(* CoDeSys 2.3 project: DPC_TM10.pro *)
(* Libraries: BODAS-design_Library_V20.lib 15.2.18 10:15:14, BODAS_RC28-14_30_Family_V01_03.lib 7.6.18 09:26:32, CIA405_Library_V02_01.lib 15.2.18 10:15:14, INEXT_Library_V01_06.lib 15.2.18 10:15:14, lib_mat.lib 15.2.18 10:15:14, RCE_InitParameter_V01_03.lib 15.2.18 10:15:14, RCE_Library_V01_03.lib 15.2.18 10:15:14, SAFOUT_Library_V02_04.lib 15.2.18 10:15:14, STANDARD_V02_00.lib 15.2.18 10:15:14, Util.lib 13.6.14 15:20:40 *)

(* Global variable list: Global_CONST *)
VAR_GLOBAL CONSTANT
	LID_DefaultSession_DU8       : USINT      := 16#7F;
	LID_DemoSession_DU8         : USINT      := 16#80;
	LID_ServiceSession_DU8      : USINT      := 16#91;
    LID_AdjustmentSession_DU8    : USINT     := 16#B3;
    LID_Adjustment1Session_DU8   : USINT     := 16#C1;
    LID_Adjustment2Session_DU8    : USINT     := 16#C2;
    LID_Adjustment3Session_DU8    : USINT    := 16#C3;
    LID_Adjustment4Session_DU8    : USINT     := 16#C4;
    LID_DevelopmentSession_DU8   : USINT     := 16#F7;


	CYCLE							: USINT	:= 10;		(* cycle time of the main task *)
	MAIN_TASK_PRIO				: BYTE	:= 100;		(*priority of the main task*)
	SIMU_motSpeed_b8			: BOOL	:= FALSE;

	DST_JOY						: INT		:= 1;			(* Type of the Drive joystick *)
	GESSMAN						: INT 	:= 0;			(* Type of the Drive joystick *)

	ST_RANGE						: INT		:= 1000;
	PAGE1_OFFSET				: INT 	:= 256;
	PAGE2_OFFSET				: INT 	:= 512;

	DELAY_STANDARD				: UINT	:= 600; 		(* increased for Fair !!! *)
	DEBOUNCE_FOR_SAVOUT		: UINT	:= 200;
	MAX_LIMIT_SPEED_MUL1000	: INT		:= 1800;
	(*LIMIT_SPEED_1_MUL1000	: INT 	:=	400;*)

	POTI_CURRENT_ERR_MIN		: INT		:= 700;		(* Unit = uA *)
	POTI_CURRENT_ERR_MAX		: INT		:= 1200;		(* Unit = uA *)

	KPDv							: REAL	:= 0.95; 	(* Volumetric efficiency *)
	(*iReductor_1					: REAL	:= 0.792;	(* передачное число редуктора МП19-4240010 *)*)

	V_TRANSM_BORDER			: INT		:= 500;		(* Граница, после которой включаются в работу моторы *)
	(*CAN1_MESSAGE_FREQ			: UINT	:= 100;		(* Промежуток между отправками посылок в шину, ms *)*)
	CYCLES_FOR_CAN_SEND		: INT		:= 10;

	Pi								: REAL	:= 3.14;		(* Число Пи *)
(******************** Definition:   PWM output - High side  *******************)
(******************************************************************************)
	POH_CL_DEBOUNCE			: UINT	:= 100;				(* debounce time [ms] for error detection *)
	POH_CL_DITHER_FREQUENCY	: UINT	:= f_100Hz_DU16;	(* dither frequency [Hz]*)
	POH_CL_RESISTANCE_MIN	: UDINT	:= 2000; 			(* min resistance of solenoid for error detection [mOhm]*)
	POH_CL_RESISTANCE_MAX	: UDINT	:= 52000;			(* max resistance of solenoid for error detection[mOhm] *)
	POH_CL_KP					: UINT	:= 250;				(*Kp factor*)
	POH_CL_KI					: UINT 	:= 250;				(*Ki factor*)
(******************** Definition:   PWM output - Low side - FAN_Drive *********)
(******************************************************************************)
	POL_CL_DEBOUNCE			: UINT	:= 100;				(* debounce time [ms] for error detection *)
	POL_CL_DITHER_FREQUENCY	: UINT	:= f_100Hz_DU16;	(* dither frequency [Hz]*)
	POL_CL_RESISTANCE_MIN	: UDINT	:= 2000; 			(* min resistance of solenoid for error detection [mOhm]*)
	POL_CL_RESISTANCE_MAX	: UDINT	:= 52000;			(* max resistance of solenoid for error detection[mOhm] *)
	POL_CL_KP					: UINT 	:= 250;				(*Kp factor*)
	POL_CL_KI					: UINT 	:= 250;				(*Ki factor*)
(******************************************************************************)
(******************** Definition:   Digital output - High side  ***************)
(******************************************************************************)
	DOH_DEBOUNCE				: UINT	:= 200;				(* debounce time [ms] for error detection *)
	DOH_DITHER_FREQUENCY		: UINT	:= f_100Hz_DU16;	(* dither frequency [Hz]*)
	DOH_RESISTANCE_MIN		: UDINT	:= 6000;				(* min resistance of solenoid for error detection [mOhm]*)
	DOH_RESISTANCE_MAX		: UDINT	:= 44000;			(* max resistance of solenoid for error detection[mOhm] *)
	DOH_WORKING_ARM_MAX		: UDINT	:= 60000;			(* Для плеч гидрораспределителя *)
	MS_IN_MINUTE				: DINT	:= 60000;

	AOV_DITHER_FREQUENCY		: UINT	:= f_100Hz_DU16;	(* dither frequency [Hz]*)

	MAX_VOLTAGE_FOR_JOY		: INT := 5000; (* Максимальное напряжение для джойстиков, мВ *)

	PWM_MODE						: INT		:= 0;					(* Режим ШИМ-выхода без поддержания тока *)
	PWM_CURRENT_MODE			: INT		:= 1;					(* Режим ШИМ-выхода с обратной связью по току *)

	AOC_MODE						: INT		:= 0;					(* Analog Output Current *)
	AOV_MODE						: INT		:= 1;					(* Analog Output Voltage *)

END_VAR

(* Global variable list: Globale_Variablen *)
VAR_GLOBAL
	para_s	: para_ts;				(* structure for the storage of the parameter *)
	err		: applError_ts;		(* structure for the error management *)
	CAN_s		: struc_Can;			(* structure for the CAN bus management *)
	J1939_s	: struc_J1939;
	IO_Chnl	: struc_IO_Chnl;		(* structure for the channels of the inputs and the outputs *)
	output	: struc_outputs;
	input		: struc_inputs;
	Uds_s    : struc_Uds;


(***********************************************************************************)
	j1939_DIESEL_DM1_s 	: j1939_dtcList_ts;
	j1939_DIESEL_DM2_s 	: j1939_dtcList_ts;
(***********************************************************************************)
	hydroDist_debounce			: UINT;				(* debounce time [ms] for error detection *)
	hydroDist_frequency			: UINT;				(* dither frequency [Hz]*)
	hydroDist_resistance_min	: UDINT; 			(* min resistance of solenoid for error detection [mOhm]*)
	hydroDist_resistance_max	: UDINT;				(* max resistance of solenoid for error detection[mOhm] *)
	hydroDist_kp_1					: UINT;				(*Kp factor*)
	hydroDist_kp_2					: UINT;				(*Kp factor*)
	hydroDist_ki_1					: UINT;				(*Ki factor*)
	hydroDist_ki_2					: UINT;				(*Ki factor*)

END_VAR

(* Global variable list: State_Machines *)
VAR_GLOBAL
	stMachine_s16				: INT		:= 0;		(*	machine state 	*)
	stStartlock_b8				: BOOL; 				(* No HW problems detected at start, if TRUE *)
	stStartAppl_b8				: BOOL;				(* Application Start condition OK, if TRUE *)
END_VAR

VAR_GLOBAL CONSTANT

(*************************************************************************************************)
	DEACTIVATED				:	INT	:=	0;
	ACTIVATED				:	INT	:=	1;

END_VAR

(* Data type in Enums *)
TYPE applError_e:
(*********************************************)
(*  DON'T MAKE ANY CHANGES TO THIS ENUMS!!   *)
(*     FILE WAS AUTOMATICALLY GENERATED!!    *)
(*********************************************)
(

   ERR_FIRST_CODE                       := 16#8000,
   ERR_CAN_DIAG                         := 16#8001,
   ERR_PWRON_SUPPLY_VB_LOW              := 16#8036,
   ERR_PWRON_SUPPLY_VSS                 := 16#8037,
   ERR_PWRON_HWMONITOR_1                := 16#8038,
   ERR_PWRON_STARTCONDITION_1           := 16#8039,
   ERR_PWRON_ENGINE_SPEED               := 16#8040,
   ERR_PWRON_HWMONITOR_2                := 16#8041,
   ERR_PWRON_STARTCONDITION_2           := 16#8042,
   ERR_PWRON_SAFOUT_CABLE_BRAKE         := 16#8043,
   ERR_PWRON_SAFOUT_SHORT_CIRCUIT       := 16#8044,
   ERR_PWRON_POWERSWITCH_1              := 16#8045,
   ERR_PWRON_POWERSUPPLY                := 16#8046,
   ERR_PWRON_POWERSWITCH_2              := 16#8047,
   ERR_PWRON_REVERSE_POWER              := 16#8048,
   ERR_PWRON_EMERGENCY_STOP             := 16#8049,
   ERR_SUPPLY_VB_HIGH                   := 16#8031,
   ERR_SUPPLY_VB_LOW                    := 16#8032,
   ERR_SUPPLY_VSS1                      := 16#8033,
   ERR_SUPPLY_VSS2                      := 16#8034,
   ERR_LAST_CODE                        := 16#8099

);
END_TYPE

(* Data type in Structures *)
TYPE applError_ts:
(***********************************************)
(*  DON'T MAKE ANY CHANGES TO THIS STRUCTURE!! *)
(*      FILE WAS AUTOMATICALLY GENERATED!!     *)
(***********************************************)
STRUCT

   First_code_b8                    : BOOL;
   Can_diag_b8                      : BOOL;
   Pwron_supply_vb_low_b8           : BOOL;
   Pwron_supply_vss_b8              : BOOL;
   Pwron_hwmonitor_1_b8             : BOOL;
   Pwron_startcondition_1_b8        : BOOL;
   Pwron_engine_speed_b8            : BOOL;
   Pwron_hwmonitor_2_b8             : BOOL;
   Pwron_startcondition_2_b8        : BOOL;
   Pwron_safout_cable_brake_b8      : BOOL;
   Pwron_safout_short_circuit_b8    : BOOL;
   Pwron_powerswitch_1_b8           : BOOL;
   Pwron_powersupply_b8             : BOOL;
   Pwron_powerswitch_2_b8           : BOOL;
   Pwron_reverse_power_b8           : BOOL;
   Pwron_emergency_stop_b8          : BOOL;
   Supply_vb_high_b8                : BOOL;
   Supply_vb_low_b8                 : BOOL;
   Supply_vss1_b8                   : BOOL;
   Supply_vss2_b8                   : BOOL;
   Last_code_b8                     : BOOL;

END_STRUCT
END_TYPE

(* Data type in Diag/Error *)
TYPE ApplErrorNew_ts :
(* ApplError_ts *)
STRUCT
	Code_u16					: UINT;
	Description_as8		: STRING(32);
(*	Description_as8		: ARRAY [1..4] OF STRING(32);*)
END_STRUCT
END_TYPE

(* Data type in Diag/Parameter *)
TYPE attr1_tu :
STRUCT
	MinValue_s16		: INT;
(*
	InputChannel_u16	: UINT;
	ListNumber_u16		: UINT;
	data_au8 			: ARRAY [1..2] OF USINT;
*)
END_STRUCT
END_TYPE

(* Data type in Diag/Parameter *)
TYPE attr2_tu :
STRUCT
	MaxValue_s16		: INT;
(*
	InputChannel_u16	: UINT;
	ListEntries_u16	: UINT;
	data_au8 			: ARRAY [1..2] OF USINT;
*)
END_STRUCT
END_TYPE

(* Data type in Diag/Parameter *)
TYPE attr3_tu :
STRUCT
	StepWidth_u16			: UINT;
(*
	FunctionNumber_u16	: UINT;
	FrequencyRange_u16	: UINT;
	data_au8 				: ARRAY [1..2] OF USINT;
*)
END_STRUCT
END_TYPE

(* Data type in Diag/Parameter *)
TYPE attr4_tu :
STRUCT
	DefaultValue_as16		: INT;
(*
	DefaultValue_as16		: ARRAY [1..16] OF INT;
	AnalogChannel_as16	: ARRAY [1..16] OF INT;
	Frequency_as16			: ARRAY [1..16] OF INT;
	data_au8 				: ARRAY [1..2] OF USINT;
*)
END_STRUCT
END_TYPE

(* Data type in Diag/Parameter *)
TYPE attr_tu :
STRUCT
	NumberOfDigits_u16	: UINT;
	BargraphMaximum_u16	: UINT;
	PostCommaDigits_u16	: UINT;
	data_au8 				: ARRAY [1..2] OF USINT;
END_STRUCT
END_TYPE

(* Data type in Diag/Parameter *)
TYPE EEPROMAdrress_ts :
STRUCT
	Page_u8		: USINT;
	IntIndex_u8	: USINT;
END_STRUCT
END_TYPE

(* Data type in 20_CAN *)
TYPE enum_Can :
	(
		CAN_RESET_STOP		:= 0,
		CAN_RESET_START	:= 1,
		CAN_RESET_WAIT		:= 2
	);
END_TYPE

(* Data type in 40_Other *)
TYPE enum_Startlock_Test :
(
	(* startlock tests *)
	TEST_SUPPLY	:= 1,
	TEST_VSS1,
	TEST_VSS2,
	TEST_VSS3,
	TEST_HWMONITOR_1,
	TEST_CONDITION_1,
	TEST_SWITCH1,
	TEST_SWITCH2,
	TEST_SAFOUT,
	TEST_DIESEL,
	TEST_HWMONITOR_2,
	TEST_CONDITION_2,
	TEST_MAX
);
END_TYPE

(* Data type in Diag/Error *)
TYPE ErrorEntry_ts :
STRUCT
	Code_u16					: UINT;
	Param_u8					: USINT;
	Frequency_u8			: USINT;
	TimeStamp_u32			: UDINT;
END_STRUCT
END_TYPE

(* Data type in Diag/Other *)
TYPE FuncParams_ts :
STRUCT
	Description_as8		: STRING(32);
(*	Description_as8		: ARRAY [1..4] OF STRING(32);*)
END_STRUCT
END_TYPE

(* Data type in Enums *)
TYPE para_e:
(*********************************************)
(*  DON'T MAKE ANY CHANGES TO THIS ENUMS!!   *)
(*    FILE WAS AUTOMATICALLY GENERATED!!     *)
(*********************************************)
(

(* Menu 1 *)

(* Basic *)
   EEP_number_1_1_1_e:= 790,      (* 0  (0 - 2) *)
   EEP_Input_to_Output_Mode_e:= 770,(* Not Active  (0 - 2) *)
   EEP_test_par_new_e:= 773,      (* Not Active  (0 - 2) *)
   EEP_test_params_e:= 771,       (* Not Active  (0 - 2) *)
   EEP_test_par2_e:= 772,         (* Not Active  (0 - 2) *)

(* Test Type *)
   EEP_Trimming_type_e:= 818,     (* 53  (0 - 511) *)
   EEP_Analog_type_e:= 819,       (* 245  (53 - ) *)
   EEP_Curve_Type_e:= 820,        (* 245  (66 - 67) *)
   EEP_Function_Type_e:= 821,     (* 248  (248 - 254) *)
   EEP_Percent_Type_e:= 822,      (* 0 % (0 - 1000) *)
   EEP_Ramp_Type_e:= 823,         (* 0 % (0 - 100) *)
   EEP_Switch_Type_e:= 824,       (* 1  ( - ) *)
   EEP_List_Type_e:= 825,         (* AOC  (3 - 2) *)

(* Test Number *)
   EEP_number_1_3_1_e:= 782,      (* 0 ms (0 - 30000) *)
   EEP_number_1_3_2_e:= 783,      (* 0 ms (0 - 30000) *)
   EEP_number_1_3_3_e:= 784,      (* 0 ms (0 - 30000) *)
   EEP_number_1_3_4_e:= 785,      (* 0 ms (0 - 30000) *)
   EEP_number_1_3_5_e:= 786,      (* 0 ms (0 - 30000) *)
   EEP_number_1_3_6_e:= 787,      (* 0 ms (0 - 30000) *)
   EEP_number_1_3_7_e:= 788,      (* 0 ms (0 - 30000) *)
   EEP_number_1_3_8_e:= 789,      (* 0 ms (0 - 30000) *)


(* Menu 2 *)

(* Output Cfg 1-8 *)
   EEP_Out_Cfg_01_e:= 832,        (* PWM  (1 - 2) *)
   EEP_Out_Cfg_02_e:= 833,        (* PWM  (1 - 2) *)
   EEP_Out_Cfg_03_e:= 834,        (* PWM  (1 - 2) *)
   EEP_Out_Cfg_04_e:= 835,        (* PWM  (1 - 2) *)
   EEP_Out_Cfg_05_e:= 836,        (* PWM  (1 - 2) *)
   EEP_Out_Cfg_06_e:= 837,        (* PWM  (1 - 2) *)
   EEP_Out_Cfg_07_e:= 838,        (* PWM  (1 - 2) *)
   EEP_Out_Cfg_08_e:= 839,        (* PWM  (1 - 2) *)

(* Output Cfg 9-16 *)
   EEP_Out_Cfg_09_e:= 840,        (* PWM  (1 - 2) *)
   EEP_Out_Cfg_10_e:= 841,        (* PWM  (1 - 2) *)
   EEP_Out_Cfg_11_e:= 842,        (* PWM  (1 - 2) *)
   EEP_Out_Cfg_12_e:= 843,        (* PWM  (1 - 2) *)
   EEP_Out_Cfg_13_e:= 844,        (* PWM  (1 - 2) *)
   EEP_Out_Cfg_14_e:= 845,        (* PWM  (1 - 2) *)
   EEP_Out_Cfg_15_e:= 846,        (* PWM  (1 - 2) *)
   EEP_Out_Cfg_16_e:= 847,        (* PWM  (1 - 2) *)

(* Output Cfg 17-24 *)
   EEP_Out_Cfg_17_e:= 848,        (* PWM  (1 - 2) *)
   EEP_Out_Cfg_18_e:= 849,        (* PWM  (1 - 2) *)
   EEP_Out_Cfg_19_e:= 850,        (* Not Active  (0 - 2) *)
   EEP_Out_Cfg_20_e:= 851,        (* Not Active  (0 - 2) *)
   EEP_Out_Cfg_21_e:= 852,        (* Not Active  (0 - 2) *)
   EEP_Out_Cfg_22_e:= 853,        (* Not Active  (0 - 2) *)
   EEP_Out_Cfg_23_e:= 854,        (* Not Active  (0 - 2) *)
   EEP_Out_Cfg_24_e:= 855,        (* Not Active  (0 - 2) *)

(* Output Cfg 25-32 *)
   EEP_Out_Cfg_25_e:= 856,        (* Not Active  (0 - 2) *)
   EEP_Out_Cfg_26_e:= 857,        (* Not Active  (0 - 2) *)
   EEP_Out_Cfg_27_e:= 858,        (* Not Active  (0 - 2) *)
   EEP_Out_Cfg_28_e:= 859,        (* Not Active  (0 - 2) *)
   EEP_Out_Cfg_29_e:= 860,        (* Not Active  (0 - 2) *)
   EEP_Out_Cfg_30_e:= 861,        (* Not Active  (0 - 2) *)
   EEP_Out_Cfg_31_e:= 862,        (* Not Active  (0 - 2) *)
   EEP_Out_Cfg_32_e:= 863,        (* Not Active  (0 - 2) *)

(* Output Cfg 33-40 *)
   EEP_Out_Cfg_33_e:= 864,        (* PWM  (2 - 2) *)
   EEP_Out_Cfg_34_e:= 865,        (* PWM  (2 - 2) *)
   EEP_Out_Cfg_35_e:= 866,        (* PWM  (2 - 2) *)
   EEP_Out_Cfg_36_e:= 867,        (* PWM  (2 - 2) *)
   EEP_Out_Cfg_37_e:= 868,        (* PWM  (1 - 2) *)
   EEP_Out_Cfg_38_e:= 869,        (* PWM  (1 - 2) *)
   EEP_Out_Cfg_39_e:= 870,        (* PWM  (1 - 2) *)
   EEP_Out_Cfg_40_e:= 871,        (* PWM  (1 - 2) *)

(* Output Cfg 41-47 *)
   EEP_Out_Cfg_41_e:= 872,        (* PWM  (1 - 2) *)
   EEP_Out_Cfg_42_e:= 873,        (* PWM  (1 - 2) *)
   EEP_Out_Cfg_43_e:= 874,        (* PWM  (1 - 2) *)
   EEP_Out_Cfg_44_e:= 875,        (* PWM  (1 - 2) *)
   EEP_Out_Cfg_45_e:= 876,        (* PWM  (1 - 2) *)
   EEP_Out_Cfg_46_e:= 877,        (* PWM  (1 - 2) *)
   EEP_Out_Cfg_47_e:= 878,        (* AOV  (3 - 2) *)

(* AOV Configuration *)
   EEP_AOV_Debounce_e:= 880,      (* 200 ms (50 - 250) *)
   EEP_AOV_Freq_e:= 881,          (* 80  (0 - 5000) *)
   EEP_AOV_Res_Min_e:= 882,       (* 0 Ohm (0 - 3000) *)
   EEP_AOV_Res_Max_e:= 883,       (* 0 Ohm (0 - 3000) *)
   EEP_AOV_Kp_e:= 884,            (* 250  (0 - 2000) *)
   EEP_AOV_Ki_e:= 885,            (* 250  (0 - 500) *)

(* AOC Configuration *)
   EEP_AOC_Debounce_e:= 888,      (* 200 ms (50 - 250) *)
   EEP_AOC_Freq_e:= 889,          (* 5000  (0 - 5000) *)
   EEP_AOC_Res_Min_e:= 890,       (* 0 Ohm (0 - 3000) *)
   EEP_AOC_Res_Max_e:= 891,       (* 0 Ohm (0 - 3000) *)
   EEP_AOC_Kp_e:= 892,            (* 250  (0 - 2000) *)
   EEP_AOC_Ki_e:= 893,            (* 250  (0 - 500) *)


(* Menu 3 *)

(* Output Value 1-8 *)
   EEP_Out_Val_01_e:= 896,        (* 0 % / mA (0 - 10000) *)
   EEP_Out_Val_02_e:= 897,        (* 0 % / mA (0 - 10000) *)
   EEP_Out_Val_03_e:= 898,        (* 0 % / mA (0 - 10000) *)
   EEP_Out_Val_04_e:= 899,        (* 0 % / mA (0 - 10000) *)
   EEP_Out_Val_05_e:= 900,        (* 0 % / mA (0 - 10000) *)
   EEP_Out_Val_06_e:= 901,        (* 0 % / mA (0 - 10000) *)
   EEP_Out_Val_07_e:= 902,        (* 0 % / mA (0 - 10000) *)
   EEP_Out_Val_08_e:= 903,        (* 0 % / mA (0 - 10000) *)

(* Output Value 9-16 *)
   EEP_Out_Val_09_e:= 904,        (* 0 % / mA (0 - 10000) *)
   EEP_Out_Val_10_e:= 905,        (* 0 % / mA (0 - 10000) *)
   EEP_Out_Val_11_e:= 906,        (* 0 % / mA (0 - 10000) *)
   EEP_Out_Val_12_e:= 907,        (* 0 % / mA (0 - 10000) *)
   EEP_Out_Val_13_e:= 908,        (* 0 % / mA (0 - 10000) *)
   EEP_Out_Val_14_e:= 909,        (* 0 % / mA (0 - 10000) *)
   EEP_Out_Val_15_e:= 910,        (* 0 % / mA (0 - 10000) *)
   EEP_Out_Val_16_e:= 911,        (* 0 % / mA (0 - 10000) *)

(* Output Value 17-36 *)
   EEP_Out_Val_17_e:= 912,        (* 0 % / mA (0 - 10000) *)
   EEP_Out_Val_18_e:= 913,        (* 0 % / mA (0 - 10000) *)
   EEP_Out_Val_33_e:= 916,        (* 0 % / mA (0 - 10000) *)
   EEP_Out_Val_34_e:= 917,        (* 0 % / mA (0 - 10000) *)
   EEP_Out_Val_35_e:= 918,        (* 0 % / mA (0 - 10000) *)
   EEP_Out_Val_36_e:= 919,        (* 0 % / mA (0 - 10000) *)

(* Output Value 37-44 *)
   EEP_Out_Val_37_e:= 920,        (* 0 % / mA (0 - 10000) *)
   EEP_Out_Val_38_e:= 921,        (* 0 % / mA (0 - 10000) *)
   EEP_Out_Val_39_e:= 922,        (* 0 % / mA (0 - 10000) *)
   EEP_Out_Val_40_e:= 923,        (* 0 % / mA (0 - 10000) *)
   EEP_Out_Val_41_e:= 924,        (* 0 % / mA (0 - 10000) *)
   EEP_Out_Val_42_e:= 925,        (* 0 % / mA (0 - 10000) *)
   EEP_Out_Val_43_e:= 926,        (* 0 % / mA (0 - 10000) *)
   EEP_Out_Val_44_e:= 927,        (* 0 % / mA (0 - 10000) *)

(* Output Value 45-47 *)
   EEP_Out_Val_45_e:= 928,        (* 0 % / mA (0 - 10000) *)
   EEP_Out_Val_46_e:= 929,        (* 0 % / mA (0 - 10000) *)
   EEP_Out_Val_47_e:= 930,        (* 0 % / mA (0 - 20000) *)

(* POH Configuration *)
   EEP_POH_Debounce_e:= 936,      (* 100 ms (50 - 250) *)
   EEP_POH_Res_Min_e:= 938,       (* 2 Ohm (0 - 3000) *)
   EEP_POH_Res_Max_e:= 939,       (* 52 Ohm (0 - 3000) *)
   EEP_POH_Kp_e:= 940,            (* 250  (0 - 2000) *)
   EEP_POH_Ki_e:= 941,            (* 250  (0 - 500) *)

(* POL Configuration *)
   EEP_POL_Debounce_e:= 944,      (* 100 ms (50 - 250) *)
   EEP_POL_Res_Min_e:= 946,       (* 2 Ohm (0 - 3000) *)
   EEP_POL_Res_Max_e:= 947,       (* 52 Ohm (0 - 3000) *)
   EEP_POL_Kp_e:= 948,            (* 250  (0 - 2000) *)
   EEP_POL_Ki_e:= 949,            (* 250  (0 - 500) *)

(* DOH Configuration *)
   EEP_DOH_Debounce_e:= 952,      (* 200 ms (50 - 250) *)
   EEP_DOH_Res_Min_e:= 954,       (* 6 Ohm (0 - 3000) *)
   EEP_DOH_Res_Max_e:= 955        (* 44 Ohm (0 - 3000) *)

);
END_TYPE

(* Data type in Structures *)
TYPE para_ts:
(***********************************************)
(*  DON'T MAKE ANY CHANGES TO THIS STRUCTURE!! *)
(*      FILE WAS AUTOMATICALLY GENERATED!!     *)
(***********************************************)
STRUCT


(* Menu 1 *)

(* Basic *)
   number_1_1_1_s16: INT;         (* 0  (0 - 2) *)
   Input_to_Output_Mode_s16: INT; (* Not Active  (0 - 2) *)
   test_par_new_s16: INT;         (* Not Active  (0 - 2) *)
   test_params_s16: INT;          (* Not Active  (0 - 2) *)
   test_par2_s16: INT;            (* Not Active  (0 - 2) *)

(* Test Type *)
   Trimming_type_s16: INT;        (* 53  (0 - 511) *)
   Analog_type_s16: INT;          (* 245  (53 - ) *)
   Curve_Type_s16: INT;           (* 245  (66 - 67) *)
   Function_Type_s16: INT;        (* 248  (248 - 254) *)
   Percent_Type_s16: INT;         (* 0 % (0 - 1000) *)
   Ramp_Type_s16: INT;            (* 0 % (0 - 100) *)
   Switch_Type_s16: INT;          (* 1  ( - ) *)
   List_Type_s16: INT;            (* AOC  (3 - 2) *)

(* Test Number *)
   number_1_3_1_s16: INT;         (* 0 ms (0 - 30000) *)
   number_1_3_2_s16: INT;         (* 0 ms (0 - 30000) *)
   number_1_3_3_s16: INT;         (* 0 ms (0 - 30000) *)
   number_1_3_4_s16: INT;         (* 0 ms (0 - 30000) *)
   number_1_3_5_s16: INT;         (* 0 ms (0 - 30000) *)
   number_1_3_6_s16: INT;         (* 0 ms (0 - 30000) *)
   number_1_3_7_s16: INT;         (* 0 ms (0 - 30000) *)
   number_1_3_8_s16: INT;         (* 0 ms (0 - 30000) *)


(* Menu 2 *)

(* Output Cfg 1-8 *)
   Out_Cfg_01_s16: INT;           (* PWM  (1 - 2) *)
   Out_Cfg_02_s16: INT;           (* PWM  (1 - 2) *)
   Out_Cfg_03_s16: INT;           (* PWM  (1 - 2) *)
   Out_Cfg_04_s16: INT;           (* PWM  (1 - 2) *)
   Out_Cfg_05_s16: INT;           (* PWM  (1 - 2) *)
   Out_Cfg_06_s16: INT;           (* PWM  (1 - 2) *)
   Out_Cfg_07_s16: INT;           (* PWM  (1 - 2) *)
   Out_Cfg_08_s16: INT;           (* PWM  (1 - 2) *)

(* Output Cfg 9-16 *)
   Out_Cfg_09_s16: INT;           (* PWM  (1 - 2) *)
   Out_Cfg_10_s16: INT;           (* PWM  (1 - 2) *)
   Out_Cfg_11_s16: INT;           (* PWM  (1 - 2) *)
   Out_Cfg_12_s16: INT;           (* PWM  (1 - 2) *)
   Out_Cfg_13_s16: INT;           (* PWM  (1 - 2) *)
   Out_Cfg_14_s16: INT;           (* PWM  (1 - 2) *)
   Out_Cfg_15_s16: INT;           (* PWM  (1 - 2) *)
   Out_Cfg_16_s16: INT;           (* PWM  (1 - 2) *)

(* Output Cfg 17-24 *)
   Out_Cfg_17_s16: INT;           (* PWM  (1 - 2) *)
   Out_Cfg_18_s16: INT;           (* PWM  (1 - 2) *)
   Out_Cfg_19_s16: INT;           (* Not Active  (0 - 2) *)
   Out_Cfg_20_s16: INT;           (* Not Active  (0 - 2) *)
   Out_Cfg_21_s16: INT;           (* Not Active  (0 - 2) *)
   Out_Cfg_22_s16: INT;           (* Not Active  (0 - 2) *)
   Out_Cfg_23_s16: INT;           (* Not Active  (0 - 2) *)
   Out_Cfg_24_s16: INT;           (* Not Active  (0 - 2) *)

(* Output Cfg 25-32 *)
   Out_Cfg_25_s16: INT;           (* Not Active  (0 - 2) *)
   Out_Cfg_26_s16: INT;           (* Not Active  (0 - 2) *)
   Out_Cfg_27_s16: INT;           (* Not Active  (0 - 2) *)
   Out_Cfg_28_s16: INT;           (* Not Active  (0 - 2) *)
   Out_Cfg_29_s16: INT;           (* Not Active  (0 - 2) *)
   Out_Cfg_30_s16: INT;           (* Not Active  (0 - 2) *)
   Out_Cfg_31_s16: INT;           (* Not Active  (0 - 2) *)
   Out_Cfg_32_s16: INT;           (* Not Active  (0 - 2) *)

(* Output Cfg 33-40 *)
   Out_Cfg_33_s16: INT;           (* PWM  (2 - 2) *)
   Out_Cfg_34_s16: INT;           (* PWM  (2 - 2) *)
   Out_Cfg_35_s16: INT;           (* PWM  (2 - 2) *)
   Out_Cfg_36_s16: INT;           (* PWM  (2 - 2) *)
   Out_Cfg_37_s16: INT;           (* PWM  (1 - 2) *)
   Out_Cfg_38_s16: INT;           (* PWM  (1 - 2) *)
   Out_Cfg_39_s16: INT;           (* PWM  (1 - 2) *)
   Out_Cfg_40_s16: INT;           (* PWM  (1 - 2) *)

(* Output Cfg 41-47 *)
   Out_Cfg_41_s16: INT;           (* PWM  (1 - 2) *)
   Out_Cfg_42_s16: INT;           (* PWM  (1 - 2) *)
   Out_Cfg_43_s16: INT;           (* PWM  (1 - 2) *)
   Out_Cfg_44_s16: INT;           (* PWM  (1 - 2) *)
   Out_Cfg_45_s16: INT;           (* PWM  (1 - 2) *)
   Out_Cfg_46_s16: INT;           (* PWM  (1 - 2) *)
   Out_Cfg_47_s16: INT;           (* AOV  (3 - 2) *)

(* AOV Configuration *)
   AOV_Debounce_s16: INT;         (* 200 ms (50 - 250) *)
   AOV_Freq_s16: INT;             (* 80  (0 - 5000) *)
   AOV_Res_Min_s16: INT;          (* 0 Ohm (0 - 3000) *)
   AOV_Res_Max_s16: INT;          (* 0 Ohm (0 - 3000) *)
   AOV_Kp_s16: INT;               (* 250  (0 - 2000) *)
   AOV_Ki_s16: INT;               (* 250  (0 - 500) *)

(* AOC Configuration *)
   AOC_Debounce_s16: INT;         (* 200 ms (50 - 250) *)
   AOC_Freq_s16: INT;             (* 5000  (0 - 5000) *)
   AOC_Res_Min_s16: INT;          (* 0 Ohm (0 - 3000) *)
   AOC_Res_Max_s16: INT;          (* 0 Ohm (0 - 3000) *)
   AOC_Kp_s16: INT;               (* 250  (0 - 2000) *)
   AOC_Ki_s16: INT;               (* 250  (0 - 500) *)


(* Menu 3 *)

(* Output Value 1-8 *)
   Out_Val_01_s16: INT;           (* 0 % / mA (0 - 10000) *)
   Out_Val_02_s16: INT;           (* 0 % / mA (0 - 10000) *)
   Out_Val_03_s16: INT;           (* 0 % / mA (0 - 10000) *)
   Out_Val_04_s16: INT;           (* 0 % / mA (0 - 10000) *)
   Out_Val_05_s16: INT;           (* 0 % / mA (0 - 10000) *)
   Out_Val_06_s16: INT;           (* 0 % / mA (0 - 10000) *)
   Out_Val_07_s16: INT;           (* 0 % / mA (0 - 10000) *)
   Out_Val_08_s16: INT;           (* 0 % / mA (0 - 10000) *)

(* Output Value 9-16 *)
   Out_Val_09_s16: INT;           (* 0 % / mA (0 - 10000) *)
   Out_Val_10_s16: INT;           (* 0 % / mA (0 - 10000) *)
   Out_Val_11_s16: INT;           (* 0 % / mA (0 - 10000) *)
   Out_Val_12_s16: INT;           (* 0 % / mA (0 - 10000) *)
   Out_Val_13_s16: INT;           (* 0 % / mA (0 - 10000) *)
   Out_Val_14_s16: INT;           (* 0 % / mA (0 - 10000) *)
   Out_Val_15_s16: INT;           (* 0 % / mA (0 - 10000) *)
   Out_Val_16_s16: INT;           (* 0 % / mA (0 - 10000) *)

(* Output Value 17-36 *)
   Out_Val_17_s16: INT;           (* 0 % / mA (0 - 10000) *)
   Out_Val_18_s16: INT;           (* 0 % / mA (0 - 10000) *)
   Out_Val_33_s16: INT;           (* 0 % / mA (0 - 10000) *)
   Out_Val_34_s16: INT;           (* 0 % / mA (0 - 10000) *)
   Out_Val_35_s16: INT;           (* 0 % / mA (0 - 10000) *)
   Out_Val_36_s16: INT;           (* 0 % / mA (0 - 10000) *)

(* Output Value 37-44 *)
   Out_Val_37_s16: INT;           (* 0 % / mA (0 - 10000) *)
   Out_Val_38_s16: INT;           (* 0 % / mA (0 - 10000) *)
   Out_Val_39_s16: INT;           (* 0 % / mA (0 - 10000) *)
   Out_Val_40_s16: INT;           (* 0 % / mA (0 - 10000) *)
   Out_Val_41_s16: INT;           (* 0 % / mA (0 - 10000) *)
   Out_Val_42_s16: INT;           (* 0 % / mA (0 - 10000) *)
   Out_Val_43_s16: INT;           (* 0 % / mA (0 - 10000) *)
   Out_Val_44_s16: INT;           (* 0 % / mA (0 - 10000) *)

(* Output Value 45-47 *)
   Out_Val_45_s16: INT;           (* 0 % / mA (0 - 10000) *)
   Out_Val_46_s16: INT;           (* 0 % / mA (0 - 10000) *)
   Out_Val_47_s16: INT;           (* 0 % / mA (0 - 20000) *)

(* POH Configuration *)
   POH_Debounce_s16: INT;         (* 100 ms (50 - 250) *)
   POH_Res_Min_s16: INT;          (* 2 Ohm (0 - 3000) *)
   POH_Res_Max_s16: INT;          (* 52 Ohm (0 - 3000) *)
   POH_Kp_s16: INT;               (* 250  (0 - 2000) *)
   POH_Ki_s16: INT;               (* 250  (0 - 500) *)

(* POL Configuration *)
   POL_Debounce_s16: INT;         (* 100 ms (50 - 250) *)
   POL_Res_Min_s16: INT;          (* 2 Ohm (0 - 3000) *)
   POL_Res_Max_s16: INT;          (* 52 Ohm (0 - 3000) *)
   POL_Kp_s16: INT;               (* 250  (0 - 2000) *)
   POL_Ki_s16: INT;               (* 250  (0 - 500) *)

(* DOH Configuration *)
   DOH_Debounce_s16: INT;         (* 200 ms (50 - 250) *)
   DOH_Res_Min_s16: INT;          (* 6 Ohm (0 - 3000) *)
   DOH_Res_Max_s16: INT;          (* 44 Ohm (0 - 3000) *)
END_STRUCT
END_TYPE

(* Data type in Diag/Other *)
TYPE ParaListEntry_ts :
STRUCT
	Description_as8		: STRING(32);
(*	Description_as8		: ARRAY [1..4] OF STRING(32);*)
END_STRUCT
END_TYPE

(* Data type in Diag/Parameter *)
TYPE Parameter_ts  :
STRUCT
	ParameterName_as8		: STRING(32);
(*	ParameterName_as8		: ARRAY [1..4] OF STRING(32);*)
	ParameterType_u8		: USINT;
	attr1_u					: INT;   	(* attr1_tu; 		MinValue_s16		: INT;	*)
	attr2_u					: INT; 		(*	attr2_tu; 		MaxValue_s16		: INT;	*)
	attr3_u					: UINT;		(* attr3_tu; 		StepWidth_u16		: UINT;	*)
	UnitCode_au8			: USINT;
(*	UnitCode_au8			: ARRAY [1..4] OF USINT;*)
	Multiplier_s16			: INT;
	Divisor_s16				: INT;
	NumberOfDigits_u16	: UINT;
	AccesslevelCode_u8	: USINT;
	attr4_u					: INT;		(* attr4_tu; 	DefaultValue_as16		: INT;	*)
	EEPROMAddress_s		: EEPROMAdrress_ts;
END_STRUCT
END_TYPE

(* Data type in Diag/Parameter *)
TYPE ParameterGroup_ts :
STRUCT
	GroupName_as8			: STRING(32);
(*	GroupName_as8			: ARRAY [1..4] OF STRING(32);*)
	Param_as					: ARRAY [1..8] OF Parameter_ts;
END_STRUCT
END_TYPE

(* Data type in Diag/Parameter *)
TYPE ParameterMenu_ts :
STRUCT
	MenuName_as8			: STRING(32);
(*	MenuName_as8			: ARRAY [1..4] OF STRING(32);*)
	ParameterGroup_as		: ARRAY [1..8] OF ParameterGroup_ts;
END_STRUCT
END_TYPE

(* Data type in Diag/ProcessValues *)
TYPE ProcessVariable_ts :
STRUCT
	ProcessVarName_as8	: STRING(32);
(*	ProcessVarName_as8	: ARRAY [1..4] OF STRING(32);*)
	ProcVarType_u8			: USINT;
	UnitCode_au8			: USINT;
(*	UnitCode_au8			: ARRAY [1..4] OF USINT;*)
	Multiplier_s16			: INT;
	Divisor_s16				: INT;
	attr_u					: UINT;		(* attr_u; 		NumberOfDigits_u16	: UINT;	*)
	AccesslevelCode_u8	: USINT;
END_STRUCT
END_TYPE

(* Data type in Diag/ProcessValues *)
TYPE ProcessVariableGroup_ts :
STRUCT
	GroupName_as8			: STRING(32);
(*	GroupName_as8			: ARRAY [1..4] OF STRING(32);*)
	ProcessVariable_as	: ARRAY [1..8] OF ProcessVariable_ts;
END_STRUCT
END_TYPE

(* Data type in 20_CAN/30_CAN_RAW *)
TYPE struc_Can :
	STRUCT
		Box			: struc_CAN_Box;   	(*structure to define the databox-numbers*)
		Id				: struc_CAN_Id;		(*structure to define the ID *)
		Chnl			: struc_CAN_Chnl;		(*structure to define the CAN channel used*)
		Data			: struc_CAN_Data;		(*storage of the data related to the CAN communication*)
		Status		: struc_CAN_Status;  (*structure to define the databox-numbers*)
		ST_LENGTH	: USINT		:= 8;
	END_STRUCT
END_TYPE

(* Data type in 20_CAN/30_CAN_RAW *)
TYPE struc_Can_Box :
STRUCT
	(*Tx_CANopen_BootUp_u16	:	UINT	:= 2;    (* Databox to transmit CANopen bootup message *)		(*для джойстика элобау - пересмотреть, возможно удалить*)*)

	Tx_Modem_201				:	UINT	:= 3;		(* first databox used for the CAN diagnostic 				*)
	Tx_Modem_202				:	UINT	:= 4;		(* second databox used for the CAN diagnostic 		*)
	Tx_Modem_203				:	UINT	:= 5;		(* the third databox used for the CAN diagnostic 	*)
	Tx_Modem_204				:	UINT	:= 6;		(*---------||------------||-----------||---------------||---------- 	*)
	Tx_Modem_205				:	UINT	:= 7;		(*---------||------------||-----------||---------------||---------- 	*)
	Tx_Modem_206				:	UINT	:= 8;		(*---------||------------||-----------||---------------||---------- 	*)
	Tx_Modem_207				:	UINT	:= 9;		(*---------||------------||-----------||---------------||---------- 	*)
	Tx_Modem_208				:	UINT	:= 10;	(*---------||------------||-----------||---------------||---------- 	*)
	Tx_Modem_209				:	UINT	:= 11;	(*---------||------------||-----------||---------------||---------- 	*)
	Tx_Modem_210				:	UINT	:= 12;
	Tx_Modem_211				:	UINT 	:= 13;
	Tx_Modem_212				:	UINT 	:= 14;
	Tx_Modem_213				:	UINT 	:= 15;
	Tx_Modem_214				:	UINT 	:= 16;
	Tx_Modem_215				:	UINT	:= 17;
	Tx_Modem_216				:	UINT	:= 18;
	Tx_MI3_220					:	UINT	:=	19;
	Tx_MI3_221					:	UINT	:=	20;
	Tx_Modem_303				:	UINT	:= 21;
	Tx_Modem_304				:	UINT	:= 22;
	Tx_Modem_305				:	UINT	:= 23;
	Tx_Modem_306				:	UINT	:= 24;
	Tx_Modem_307				:	UINT	:= 25;
	Tx_Modem_308				:	UINT	:= 26;
	Tx_Modem_309				:	UINT	:= 27;
	Tx_Modem_310				:	UINT	:= 28;
	Tx_Modem_311				:	UINT	:= 29;
	Tx_Modem_401				:	UINT	:= 30;		(* сообщение об ошибках 1-64*)
	Tx_Modem_402				:	UINT	:= 31;		(* сообщение об ошибках 65-99*)
	Tx_Topcon					:	UINT	:= 32;
	Tx_TSC_Cummins				:	UINT	:= 33;
	Tx_TSC_YaMZ					:	UINT	:= 34;
	Tx_DieselPoti				:	UINT	:= 35;
	Tx_DM1_Diesel				:	UINT	:= 36;
	Tx_Modem_405				:	UINT	:= 37;		(* сообщение о сохраненных ошибках 1-64*)
	Tx_Modem_406				:	UINT	:= 38;		(* сообщение о сохраненных ошибках 65-99*)
	Tx_DM2_Diesel				:	UINT	:= 39;
	Tx_Req_PGN_from_Dies		:	UINT	:= 40;		(* Запрос ошибок от ДВС *)
	Tx_Req_DM3_Cummins		:	UINT	:= 41;		(* Запрос на удаление ошибок ДВС Cummins *)
(******************************************************************************)
(******************** Definition: databoxes RX  *******************************)
(******************************************************************************)
(*Rx_BODAS1				: UINT	:= 1;		used BY BODAS Diag*)
(*Rx_BODAS2				: UINT	:= 2;		used BY BODAS Diag*)
	Rx_HG405_u16				:	UINT	:= 3;		(* used to receive CAN from drive / steer joystick *)
	Rx_Elobau_A_u16			:	UINT	:= 4;		(* used to receive CAN from drive / steer joystick *)
	Rx_Elobau_B_u16			:	UINT	:= 5;		(* used to receive CAN from joy buttons *)
	Rx_RemoteControl_A_u16	:	UINT	:= 6;		(* Пульт дистанционного управления *)
	Rx_RemoteControl_B_u16	:	UINT	:= 7;		(* Пульт дистанционного управления *)
	Rx_RemoteControl_C_u16	:	UINT	:= 8;	(* Пульт дистанционного управления *)
	Rx_AZK_u16					:	UINT	:= 9;
	Rx_Attach_KVG				:	UINT	:= 10;
	Rx_Modem_300				:	UINT	:= 11;
	Rx_Modem_301				:	UINT	:= 12;
	Rx_PosSensBlade			:	UINT	:= 13;
	Rx_PosSensChassis			:	UINT	:= 14;
	Rx_PosSensRipper			:	UINT	:= 15;
	Rx_JoyAttach				:	UINT	:= 16;
	Rx_DieselPoti				:	UINT	:= 17;
	Rx_GpsRover					:	UINT	:= 18;
	Rx_Topcon					:	UINT	:= 19;
	Rx_Start_Stop_Button		:	UINT	:= 20;
END_STRUCT
END_TYPE

(* Data type in 20_CAN/10_General CAN *)
TYPE struc_Can_Chnl :
	STRUCT
		(* can bus interfaces *)
		BODAS_SERVICE_u8		: USINT		:= CAN_1;  	(* Bodas Service, Should not be changed - always CAN1  !!! *)
		CANALYZER_u8			: USINT		:= CAN_1;	(*CAN bus used for the communication with BODAS-service*)
		J1939_DIESEL_u8		: USINT		:= CAN_1;	(* CAN bus used for communication with diesel engine*)
		JOYSTICKS_u8			: USINT		:= CAN_1;	(* CAN bus used for communication with HG405 joystick*)
		CAN_modem_u8			: USINT		:=	CAN_1;	(* CAN bus used for communication with CAN_modem *)
		Remote_Control_u8		: USINT		:=	CAN_1;	(* Пульт дистанционного управления *)
		Attachments_KVG_u8	: USINT		:=	CAN_1;	(* Плата управления навесным оборудованием КВГ *)
		AZK_u8					: USINT		:=	CAN_1;	(* Прием посылок от АЗК - монитор Bosch *)
		ELOBAU_u8				: USINT		:= CAN_1;	(*  *)
		Position_Sensors		: USINT		:= CAN_1;
	END_STRUCT
END_TYPE

(* Data type in 20_CAN/30_CAN_RAW *)
TYPE struc_Can_Data :
STRUCT
	(* @CAN *)
  (*CAN1_Rx_buf				: ARRAY [1..20] OF can_Message_ts;		(* can receive buffer - NOT NEEDED AS in BD is DONE BY API!	*)
  CAN1_Tx_buf				: ARRAY [1..20] OF can_Message_ts;		(* can send buffer  	- NOT NEEDED AS in BD is DONE BY API! *)*)

	(* Tx data buffer *)
	(*can_1_TxBuf_as				: ARRAY [1..2] OF can_Message_ts;*)
	(*TxOperationalStatus_au8	: ARRAY [1..8] OF USINT;	(*storage of the data for the diagnostic *)*)

	can_TxMsg_as				: ARRAY [1..41] OF can_TxDatabox_ts;		(* can tx msg boxes *)

	RxHG405_au8					: ARRAY [1..8] OF USINT;   (* data buffer for HG405 joystick *)
	RxElobau_A_au8				: ARRAY [1..8] OF USINT;   (* data buffer for HG405 joystick *)
	RxElobau_B_au8				: ARRAY [1..8] OF USINT;   (* data buffer for HG405 joystick *)

	RxJoyAttachDst				: ARRAY [1..8] OF USINT;

	RxRemoteControl_A_au8	: ARRAY [1..8] OF USINT;	 (* Данные от пульта дистанционного управления *)
	RxRemoteControl_B_au8	: ARRAY [1..8] OF USINT;	 (* Данные от пульта дистанционного управления *)
	RxRemoteControl_C_au8	: ARRAY [1..8] OF USINT;	 (* Данные от пульта дистанционного управления *)

	RxAttachmentsKVG_au8		: ARRAY [1..8] OF USINT;
	RxAZK							: ARRAY [1..8] OF USINT;

	RxModem_300_au8			: ARRAY [1..8] OF USINT;	(* storage of the data for the CAN-modem *)
	RxModem_301_au8			: ARRAY [1..8] OF USINT;	(* storage of the data for the CAN-modem *)

	(**Position Sensors**)
	RxPosSensBlade				: ARRAY [1..8] OF USINT;
	RxPosSensChassis			: ARRAY [1..8] OF USINT;
	RxPosSensRipper			: ARRAY [1..8] OF USINT;
	RxGpsRover					: ARRAY [1..8] OF USINT;

	RxStartStopButton			: ARRAY [1..8] OF USINT;	(* Блок пуска-глушения *)
(*************--Tx--*************)
	TxModem_201_au8			: ARRAY [1..8] OF USINT;	(* storage of the data for the CAN-modem *)
	TxModem_202_au8			: ARRAY [1..8] OF USINT;	(* storage of the data for the CAN-modem *)
	TxModem_203_au8			: ARRAY [1..8] OF USINT;	(* storage of the data for the CAN-modem *)
	TxModem_204_au8			: ARRAY [1..8] OF USINT;	(* storage of the data for the CAN-modem *)
	TxModem_205_au8			: ARRAY [1..8] OF USINT;	(* storage of the data for the CAN-modem *)
	TxModem_206_au8			: ARRAY [1..8] OF USINT;	(* storage of the data for the CAN-modem *)
	TxModem_207_au8			: ARRAY [1..8] OF USINT;	(* storage of the data for the CAN-modem *)
	TxModem_208_au8			: ARRAY [1..8] OF USINT;	(* storage of the data for the CAN-modem *)
	TxModem_209_au8			: ARRAY [1..8] OF USINT;	(* storage of the data for the CAN-modem *)
	TxModem_210_au8			: ARRAY [1..8] OF USINT;	(* storage of the data for the CAN-modem *)
	TxModem_211_au8			: ARRAY [1..8] OF USINT;	(* storage of the data for the CAN-modem *)
	TxModem_212_au8			: ARRAY [1..8] OF USINT;	(* storage of the data for the CAN-modem *)
	TxModem_213_au8			: ARRAY [1..8] OF USINT;	(* storage of the data for the CAN-modem *)
	TxModem_214_au8			: ARRAY [1..8] OF USINT;	(* storage of the data for the CAN-modem *)
	TxModem_215_au8			: ARRAY [1..8] OF USINT;	(* storage of the data for the CAN-modem *)
	TxModem_216_au8			: ARRAY [1..8] OF USINT;	(* storage of the data for the CAN-modem *)

	TxMI3_220_au8				: ARRAY [1..8] OF USINT;	(* storage of the data for the MI-3 *)
	TxMI3_221_au8				: ARRAY [1..8] OF USINT;	(* storage of the data for the MI-3 *)
	(* Актуальные ошибки контроллера ГСТ *)
	TxModem_401_au8			: ARRAY [1..8] OF USINT;
	TxModem_402_au8			: ARRAY [1..8] OF USINT;
	(* Сохраненные ошибки контроллера ГСТ *)
	TxModem_405_au8			: ARRAY [1..8] OF USINT;
	TxModem_406_au8			: ARRAY [1..8] OF USINT;

	TxModem_303_au8			: ARRAY [1..8] OF USINT;	(* storage of the data for the CAN-modem *)
	TxModem_304_au8			: ARRAY [1..8] OF USINT;	(* storage of the data for the CAN-modem *)
	TxModem_305_au8			: ARRAY [1..8] OF USINT;	(* storage of the data for the CAN-modem *)
	TxModem_306_au8			: ARRAY [1..8] OF USINT;	(* storage of the data for the CAN-modem *)
	TxModem_307_au8			: ARRAY [1..8] OF USINT;	(* storage of the data for the CAN-modem *)
	TxModem_308_au8			: ARRAY [1..8] OF USINT;	(* storage of the data for the CAN-modem *)
	TxModem_309_au8			: ARRAY [1..8] OF USINT;	(* storage of the data for the CAN-modem *)
	TxModem_310_au8			: ARRAY [1..8] OF USINT;	(* storage of the data for the CAN-modem *)
	TxModem_311_au8			: ARRAY [1..8] OF USINT;	(* storage of the data for the CAN-modem *)
	(*TxRemoteControl_au8	: ARRAY	[1..8] OF USINT;	 (* Данные передаваемые на пульт дистанционного управления *)*)

	(* Topcon *)
	Rx_Topcon_au8				: ARRAY [1..8] OF USINT;
	Tx_Topcon_au8				: ARRAY [1..8] OF USINT;
	(* Engines *)
	TxTscCummins				: ARRAY [1..8] OF USINT;	(* Посылка с требуемой скоростью вращения для Cummins *)
	TxTscYaMZ					: ARRAY [1..8] OF USINT;	(* Посылка с требуемой скоростью вращения для ЯМЗ *)
	(* Ручка газа *)
	RxDiesPoti					: ARRAY [1..8] OF USINT;
	TxDiesPoti					: ARRAY [1..8] OF USINT;
	(* Сообщение с ошибками ДВС для дисплея *)
	Tx_DM1_Diesel_au8			: ARRAY [1..8] OF USINT;
	Tx_DM2_Diesel_au8			: ARRAY [1..8] OF USINT;
	Tx_Req_PGN_au8				: ARRAY [1..8] OF USINT;
	Tx_DM3_Cummins_au8		: ARRAY [1..8] OF USINT;


	Databox_data_1				: ARRAY [1..8] OF USINT;
	Databox_data_2				: ARRAY [1..8] OF USINT;
	Databox_data_3				: ARRAY [1..8] OF USINT;
	Databox_data_4				: ARRAY [1..8] OF USINT;
END_STRUCT
END_TYPE

(* Data type in 20_CAN/30_CAN_RAW *)
TYPE struc_Can_Id :
	STRUCT
(******************************************************************************)
(******************** Definition: CAN IDs  ************************************)
(******************************************************************************)
		Rx_HG405						: 	UINT := 	16#2FE;			(* Define receive HG405 joystick identifier *)

		Rx_AttachDstJoy			: 	UINT := 	16#180;			(* Джойстик управления навесным оборудованием, ДСТ *)

		Rx_Elobau_A_u16			: 	UINT := 	16#190;			(* Define receive Elobau joystick identifier *)
		Rx_Elobau_B_u16			: 	UINT := 	16#290;			(* Define receive Elobau joystick identifier *)

		Rx_RemoteControl_A_u16	:	UINT :=	16#195;			(* ПДУ - джойстик движения 						*)
		Rx_RemoteControl_B_u16	:	UINT :=	16#196;			(* ПДУ - джойстик навесного						*)
		Rx_RemoteControl_C_u16	:	UINT :=	16#198;			(* ПДУ - обороты ДВС									*)
		(*Tx_RemoteControl_u16		:	UINT :=	16#199;*)

		Rx_Attachments_KVG_u16	:	UINT :=	16#199;			(* Плата управления навесным оборудованием КВГ *)

		(*Посылка 501 - от преобразователя K-Line/CAN идет к монитору АЗК Bosch *)
		Rx_AZK_d32					:	DINT :=	16#18050203;	(* Прием посылок от АЗК - монитор Bosch *)
		(* Датчики положения отвала/рамы/рыхлителя *)
		Rx_Pos_Sens_Blade			:	DINT :=	16#18050603;
		Rx_Pos_Sens_Chassis		:	DINT :=	16#18050703;
		Rx_Pos_Sens_Ripper		:	DINT :=	16#18050803;
		Rx_GPS_Rover				:	DINT :=	16#18051003;	(* Модем *)

		Rx_Start_Stop_Button		:	DINT :=	16#1802BD03;	(* Блок пуска-глушения *)

		Tx_Modem_201				:	DINT :=	16#18020103;
		Tx_Modem_202				:	DINT :=	16#18020203;
		Tx_Modem_203				:	DINT :=	16#18020303;
		Tx_Modem_204				:	DINT :=	16#18020403;
		Tx_Modem_205				:	DINT :=	16#18020503;
		Tx_Modem_206				:	DINT :=	16#18020603;
		Tx_Modem_207				:	DINT :=	16#18020703;
		Tx_Modem_208				:	DINT :=	16#18020803;
		Tx_Modem_209				:	DINT :=	16#18020903;
		Tx_Modem_210				:	DINT :=	16#18021003;
		Tx_Modem_211				:	DINT :=	16#18021103;
		Tx_Modem_212				:	DINT :=	16#18021203;
		Tx_Modem_213				:	DINT :=	16#18021303;
		Tx_Modem_214				:	DINT :=	16#18021403;
		Tx_Modem_215				:	DINT :=	16#18021503;
		Tx_Modem_216				:	DINT :=	16#18021603;

		Tx_MI3_220					:	DINT :=	16#18022003;
		Tx_MI3_221					:	DINT :=	16#18022103;

		Rx_Modem_300				:	DINT :=	16#18030003;
		Rx_Modem_301				:	DINT :=	16#18030103;

		Tx_Modem_303				:	DINT :=	16#18030303;
		Tx_Modem_304				:	DINT :=	16#18030403;
		Tx_Modem_305				:	DINT :=	16#18030503;
		Tx_Modem_306				:	DINT :=	16#18030603;
		Tx_Modem_307				:	DINT :=	16#18030703;
		Tx_Modem_308				:	DINT :=	16#18030803;
		Tx_Modem_309				:	DINT :=	16#18030903;
		Tx_Modem_310				:	DINT :=	16#18031003;
		Tx_Modem_311				:	DINT :=	16#18031103;
		(* Актуальные ошибки контроллера ГСТ *)
		Tx_Modem_401				:	DINT :=	16#18040103;
		Tx_Modem_402				:	DINT :=	16#18040203;
		(* Сохраненные ошибки контроллера ГСТ *)
		Tx_Modem_405				:	DINT :=	16#18040503;
		Tx_Modem_406				:	DINT :=	16#18040603;
		(* Topcon *)
		Rx_Topcon					:	DINT :=	16#0CEF8047;
		Tx_Topcon					:	DINT :=	16#18F00D80;
		(* Двигатели *)
		Tx_TSC_Cummins				:	DINT :=	16#0C000007;
		Tx_TSC_YaMZ					:	DINT :=	16#0C000024;	(* Проверить *)
		(* Ручка газа *)
		Rx_DieselPoti				:	DINT :=	16#18018919;
		Tx_DieselPoti				:	DINT :=	16#18018803;
		(* Сообщение с ошибками ДВС для дисплея *)
		Tx_DM1_Diesel				:	DINT :=	16#18FFA003;
		Tx_DM2_Diesel				:	DINT :=	16#18FFA303;


		Tx_Req_PGN					:	DWORD :=	16#18EA0000;	(* Подготовка для расчета ID для запроса PGN у двигателя *)
	END_STRUCT
END_TYPE

(* Data type in 20_CAN/10_General CAN *)
TYPE struc_Can_Status :
STRUCT

(*@CAN*)

	BODAS_SERVICE_u16	: UINT;
	BUS2_u16				: UINT;
	BUS3_u16				: UINT;
	Channel_CAN_1		: UINT;
(******************************************************************************)
(******************** Status: databoxes TX  ***********************************)
(******************************************************************************)
	(*CAN_modem_201_u16	: UINT;		(* state of the first databox used for the CAN diagnostic *)
	CAN_modem_202_u16	: UINT;		(* state of the second databox used for the CAN diagnostic *)
	CAN_modem_203_u16	: UINT;		(* state of the second databox used for the CAN diagnostic *)
 	CAN_modem_204_u16	: UINT;		(* state of the first databox used for the CAN diagnostic *)
	CAN_modem_205_u16	: UINT;		(* state of the second databox used for the CAN diagnostic *)
	CAN_modem_206_u16	: UINT;		(* state of the second databox used for the CAN diagnostic *)
	CAN_modem_207_u16	: UINT;		(* state of the second databox used for the CAN diagnostic *)
	CAN_modem_208_u16	: UINT;		(* state of the second databox used for the CAN diagnostic *)
	CAN_modem_209_u16	: UINT;		(* state of the second databox used for the CAN diagnostic *)
	CAN_modem_210_u16	: UINT;		(* state of the second databox used for the CAN diagnostic *)
	CAN_modem_211_u16	: UINT;		(* state of the second databox used for the CAN diagnostic *)
	CAN_modem_212_u16	: UINT;		(* state of the second databox used for the CAN diagnostic *)
	CAN_modem_213_u16	: UINT;		(* state of the second databox used for the CAN diagnostic *)
	CAN_modem_214_u16	: UINT;		(* state of the second databox used for the CAN diagnostic *)
	CAN_modem_215_u16	: UINT;		(* state of the second databox used for the CAN diagnostic *)
	CAN_modem_216_u16	: UINT;		(* state of the second databox used for the CAN diagnostic *)*)

	(*MI3_220_u16			: UINT;		(* МИ-3 *)
	MI3_221_u16			: UINT;		(* МИ-3 *)

	CAN_modem_401_u16	: UINT;		(* state of the second databox used for the CAN diagnostic*)
	CAN_modem_402_u16	: UINT;		(* state of the second databox used for the CAN diagnostic*)*)
(******************************************************************************)
(******************** Status: databoxes RX  ***********************************)
(******************************************************************************)
	HG405_u16				: UINT;
	Elobau_A_u16			: UINT;
	Elobau_B_u16			: UINT;
	EEC1_u16					: UINT;		(*state of the databox used to receive values from the customer*)
	(*EEC2_u16					: UINT;		(*state of the databox used to receive values from the customer*)
	EEC3_u16					: UINT;		(*state of the databox used to receive values from the customer*)*)
	ET1_u16					: UINT;
	EFL_u16					: UINT;
	IC1_u16					: UINT;
	TFAC_u16					: UINT;
	RemoteControl_A_u16	: UINT;		(* Пульт дистанционного управления *)
	RemoteControl_B_u16	: UINT;		(* Пульт дистанционного управления *)
	RemoteControl_C_u16	: UINT;		(* Пульт дистанционного управления *)
	Attachments_KVG		: UINT;
	AZK						: UINT;
	Modem_300				: UINT;
	Modem_301				: UINT;
	(*********)
	PosSensBlade			: UINT;
	PosSensChassis			: UINT;
	PosSensRipper			: UINT;
	GpsRover					: UINT;
	(*********)
	JoyAttachDST			: UINT;
	DieselPoti				: UINT;
	(**)
	LevelingTopcon			: UINT;
	DM1_Diesel_u16			: UINT;
	DM2_Diesel_u16			: UINT;

	Start_Stop_Btn_u16	: UINT;		(* Блок пуска-глушения *)
END_STRUCT
END_TYPE

(* Data type in 10_IO *)
TYPE struc_inputs :
STRUCT

	potiDriveCAN_s16			: INT;  	(* Speed Setpoint with deadbnd (CAN part), [ -1000, 1000], Unit = 0.1% *)
	potiSteerCAN_s16			: INT;	(* Steer Setpoint with deadband (CAN part), [ -1000, 1000], Unit = 0.1% *)
	potiDriveCAN_raw_s16		: INT;	(* Speed Setpoint (CAN part), [ -1000, 1000], Unit = 0.1% *)
	potiSteerCAN_raw_s16		: INT;	(* Steer Setpoint (CAN part), [ -1000, 1000], Unit = 0.1% *)
	potiDriveANA_s16			: INT;	(* Speed Setpoint (Analog part), [ -1000, 1000], Unit = 0.1% *)
	iDriveANA_uA_s16			: INT; 	(* Current through drive poti, Unit = 1/1000 mA *)
	potiSteerANA_s16			: INT;	(* Steer Setpoint (Analog part), [ -1000, 1000], Unit = 0.1% *)
	iSteerANA_uA_s16			: INT; 	(* Current through steer poti, Unit = 1/1000 mA *)
	potiDriveANA_raw_s16		: INT;	(* Speed Setpoint (Analog part), [ -1000, 1000], Unit = 0.1% w/o deadband *)
	potiSteerANA_raw_s16		: INT;	(* Steer Setpoint (Analog part), [ -1000, 1000], Unit = 0.1% w/o deadband *)

	potiDriveSet_s16			: INT;	(* Drive averaged Setpoint, [ -1000, 1000], Unit = 0.1% *)
	potiSteerSet_s16			: INT;	(* Steer averaged Setpoint, [ -1000, 1000], Unit = 0.1% *)
(**********************************************************************************************************)
(***************************** Пульт дистанционного управления ********************************************)
(**********************************************************************************************************)
	potiDrive_RC_s16			: INT;	(* Управление движением 								*)
	potiSteer_RC_s16			: INT;  	(* Управление рулением 									*)
	potiDir_RC_s16				: INT;	(* Управление навесным оборудованием				*)
	potiSide_RC_s16			: INT;	(* Управление навесным оборудованием				*)
	btn_GearUp_RC_b8			: BOOL;	(* Уменьшение скорости									*)
	btn_GearDn_RC_b8			: BOOL;	(* Увеличение скорости									*)
	btn_EquipMode_RC_b8		: BOOL;	(* Выбор режима оборудования							*)
	btn_SwimMode_RC_b8		: BOOL;	(* Включение "плавающего"								*)
	btn_A_RC_b8					: BOOL;	(* Дополнительная кнопка на джойстике навесного	*)
	potiDiesel_RC_s16			: INT;	(* Обороты ДВС												*)

END_STRUCT
END_TYPE

(* Data type in 10_IO *)
TYPE struc_IO_Chnl :
STRUCT
(******************** Definition: Input channel *************************************)

(******************** 	Frequency Inputs 					*************************************)
	FI_IDR_DIESEL				:	UDINT	:=	IN_69_FI;			(* Обороты вращения дизеля 		*)

	FI_HDD_MOTOR_L				:	UDINT	:=	IN_66_FI;			(* 3х-проводный датчик скорости 	*)
	FI_HDD_MOTOR_R				:	UDINT	:=	IN_67_FI;			(* 3х-проводный датчик скорости 	*)
	FI_DSM_MOTOR_L				:	UDINT	:=	IN_71_FI;			(* 2х-проводный датчик скорости 	*)
	FI_DSM_MOTOR_R				:	UDINT	:=	IN_72_FI;			(* 2х-проводный датчик скорости	*)
(******************** 	Digital Inputs 						*************************************)
	AID_EQUIP_MODE				:	UDINT	:=	IN_1_AIV;			(* Выбор режима оборудования 			*)
	AID_SWIM_MODE				:	UDINT	:=	IN_2_AIV;			(* Включение "плавающего" 				*)
	AID_BUTTON_B				:	UDINT	:=	IN_3_AIV;			(* Доп. функционал на кнопке B	 	*)
	AID_BUTTON_A				:	UDINT	:=	IN_5_AIV;			(* Доп. функционал на кнопке A 		*)

	AID_NON_SIGNAL				:	UDINT := IN_4_AIV;			(* Выключение сигнала заднего хода	*)
	AID_OPERATOR_SENS			:	UDINT := IN_6_AIV;			(* Датчик присутствия оператора		*)
	AID_PARKING_SWT			:	UDINT	:= IN_7_AIV;			(* Включатель парковочного режима	*)
	AID_SAFETY					:	UDINT	:=	IN_10_AIV; 			(* Выключатель безопасности 			*)
	AID_TOWING 					:	UDINT	:= IN_11_AIV;			(* Включение транспортирования 		*)
	AID_BOM_SWITCH				:	UDINT := IN_12_AIV;			(* Включение режима ВОМ 				*)
	AID_FAN_SWITCH				:	UDINT := IN_13_AIV;			(* Переключение режима FANDrive 		*)
	AID_BOM_REV					:	UDINT	:=	IN_14_AIV;			(* Реверс ВОМ 								*)
	AID_FAN_REV					:	UDINT :=	IN_16_AIV;			(* Включение реверса FANDrive 		*)
	AID_PEDAL_MODE				:	UDINT	:= IN_20_AIV;			(* Переключение режима инч-педали	*)
	AID_START_DIESEL			:	UDINT	:=	IN_23_AIV;			(* Запуск дизеля 							*)
	AID_CLOSE_CRANE			:	UDINT	:=	IN_24_AIV;			(* Датчик крана гидробака				*)
(******************** 	Analog Inputs 						*************************************)
	AI_TEMP_ENVIR				:	UDINT	:=	IN_15_AIV;			(* Темп-ра окружающей среды 			*)

	AI_HYD_PUMP_L				:	UDINT	:=	IN_25_AIV;			(* Датчик давления левого борта					*)
	AI_HYD_PUMP_R				:	UDINT	:=	IN_26_AIV;			(* Датчик давления правого борта 				*)
	AI_HYD_BRAKE				:	UDINT	:=	IN_27_AIV;			(* Давление растормаживания						*)
	AI_HYD_ATT_PUMP			:	UDINT	:=	IN_28_AIV;			(* Давление в контуре навесного оборудования	*)
	AI_HYD_FAN_PUMP			:	UDINT	:=	IN_29_AIV;			(* Давление в контуре FAN-drive					*)

	AI_BRAKE_PEDAL				:	UDINT	:=	IN_33_AIV;			(* Датчик педали дисселератора 		*)
	AI_TEMP_AIR					:	UDINT	:=	IN_34_AIV;			(* Темп-ра воздуха турбины 			*)
	AI_BOM_SPEED				:	UDINT	:=	IN_37_AIV;			(* Обороты вращения ВОМ 				*)
	AI_POTI_DIESEL				:	UDINT	:=	IN_39_AIV;			(* Датчик положения рейки 				*)
	AI_TEMP_OIL					:	UDINT	:=	IN_40_AIV;			(* Темп-ра масла трансмиссии 			*)
	AI_TEMP_COOLANT			:	UDINT	:=	IN_41_AIV;			(* Темп-ра охлаждающей жидкости		*)

	AI_JOY_DRIVE				:	UDINT	:=	IN_52_AIV;			(* Потенциометр движения				*)
	AI_JOY_STEER				:	UDINT	:=	IN_53_AIV;			(* Потенциометр руления 				*)
	AI_JOY_DRIVE_CM			:	UDINT	:=	IN_54_AIC;
	AI_JOY_STEER_CM			:	UDINT	:=	IN_55_AIC;

	(*AI_JOY_DIRECTION_CM 		:	UDINT := IN_56_AIC;			(* Токовый вход джойстик навесного  *)
	AI_JOY_SIDE_CM				:	UDINT :=	IN_57_AIC;			(* Токовый вход джойстик навесного  *)*)
	AI_JOY_DIRECTION			:	UDINT	:=	IN_58_AIV;			(* Джойстик Вперед/Назад навесного	*)
	AI_JOY_SIDE					:	UDINT	:=	IN_59_AIV;			(* Джойстик Влево/Вправо навесного	*)
(********************		Sensors Inputs 						*************************************)
	DI_SENS_1					:	UDINT	:=	IN_43_DI;			(* Датчик низкого давления масла ДВС - 86	 *)
	DI_SENS_2					:	UDINT	:=	IN_44_DI;			(* Датчик перегрева масла в баке 	 -	T°	 *)
	DI_SENS_3					:	UDINT	:=	IN_45_DI;			(* Датчик засора топливного фильтра  - 16	 *)
	DI_SENS_4					:	UDINT	:=	IN_46_DI;			(* Датчик неисправности НШ 			 - НШ	 *)
	DI_SENS_5					:	UDINT	:=	IN_47_DI;			(* Датчик засора фильтра навесного	 - ЗФН *)
	DI_SENS_6					:	UDINT	:=	IN_48_DI;			(* Датчик засор фильтра насосов ГСТ	 - 106 *)
	DI_SENS_7					:	UDINT	:=	IN_49_DI;			(* Датчик засор воздушного фильтра	 - ЗФВ *)
	DI_SENS_8					:	UDINT	:=	IN_50_DI;			(* Датчик низкий уровень гидробака	 - 213 *)
	DI_SENS_9					:	UDINT	:=	IN_51_DI;			(* Датчик низкий уровень топлива		 - 125 *)
(******************** 	Definition: Output channel ************************************)
	POH_PUMP_FORW_L			:	UDINT	:=	OUT_1_POH_CL;		(* Левый борт Вперед		*)
	PIC_PUMP_FORW_L			:	UDINT	:=	OUT_1_PIC;			(* Левый борт Вперед		*)
	POH_PUMP_REV_L				:	UDINT	:=	OUT_2_POH_CL;		(* Левый борт Назад		*)
	PIC_PUMP_REV_L				:	UDINT	:=	OUT_2_PIC;			(* Левый борт Назад		*)
	POH_PUMP_FORW_R			:	UDINT	:=	OUT_3_POH_CL;		(* Правый борт Вперед	*)
	PIC_PUMP_FORW_R			:	UDINT	:=	OUT_3_PIC;			(* Правый борт Вперед	*)
	POH_PUMP_REV_R				:	UDINT	:=	OUT_4_POH_CL;		(* Правый борт Назад 	*)
	PIC_PUMP_REV_R				:	UDINT	:=	OUT_4_PIC;			(* Правый борт Назад 	*)
	POH_MOTOR_L					:	UDINT	:=	OUT_5_POH_CL;		(* Левый мотор 			*)
	PIC_MOTOR_L					:	UDINT	:=	OUT_5_PIC;			(* Левый мотор 			*)
	POH_MOTOR_R					:	UDINT	:=	OUT_6_POH_CL;		(* Правый мотор 			*)
	PIC_MOTOR_R					:	UDINT	:=	OUT_6_PIC;			(* Правый мотор 			*)

	POL_GIDRO_FWD				:	UDINT	:=	OUT_37_POL_CL;		(* Навесное оборудование. Вперед.*)
	PIC_GIDRO_FWD				:	UDINT	:=	OUT_37_PIC;			(* Навесное оборудование. Вперед.*)
	POL_GIDRO_REV				:	UDINT	:=	OUT_38_POL_CL;		(* Навесное оборудование. Назад 	*)
	PIC_GIDRO_REV				:	UDINT	:=	OUT_38_PIC;			(* Навесное оборудование. Назад 	*)
	POL_GIDRO_L					:	UDINT	:=	OUT_41_POL_CL;		(* Навесное оборудование. Влево 	*)
	PIC_GIDRO_L					:	UDINT	:=	OUT_41_PIC;			(* Навесное оборудование. Влево 	*)
	POL_GIDRO_R					:	UDINT	:=	OUT_42_POL_CL;		(* Навесное оборудование. Вправо *)
	PIC_GIDRO_R					:	UDINT	:=	OUT_42_PIC;			(* Навесное оборудование. Вправо *)

	DOH_WORK_MODE_1			:	UDINT	:= OUT_19_DOH;			(* Режим "Бульдозер" 					*)
	DOH_WORK_MODE_2			:	UDINT	:= OUT_20_DOH;			(* Режим "Рыхлитель" 					*)

	DOH_BRAKES					:	UDINT	:= OUT_23_DOH;			(* Клапан растормаживания 				*)
	PIC_BRAKES					:	UDINT	:= OUT_23_PIC;			(* Клапан растормаживания 				*)

	DOH_IND_REVERS				:	UDINT	:= OUT_26_DOH;			(* Индикатор движения задним ходом	*)
	DOH_START_DIESEL			:	UDINT	:=	OUT_28_DOH;			(* Выход запуска дизеля 				*)
	DOH_FLASHING_BEACON		:	UDINT := OUT_29_DOH;			(* Маяк 										*)
	DOH_CONT_BAL_VALVE		:	UDINT	:= OUT_30_DOH;			(* Клапан блокировки контргруза *)

	POL_FAN_DRIVE				:	UDINT	:=	OUT_39_POL_CL;		(* Клапан FANdrive 						*)
	PIC_FAN_DRIVE				:	UDINT	:=	OUT_39_PIC;			(* Клапан FANdrive 						*)

	POL_OPTION_BOM				:	UDINT	:=	OUT_40_POL_CL;		(* ВОМ или другая опция 				*)
	PIC_OPTION_BOM				:	UDINT	:=	OUT_40_PIC;			(* ВОМ или другая опция 				*)
(***************************************************************************************)
(*Сейчас не реализован вариант установки трехпозиционного отвала на старую кабину*)

	DOH_REV_FANDRV				:	UDINT	:= OUT_21_DOH;			(* Клапан реверса FAN Drive			*)
	DOH_IDLE_FANDRV			:	UDINT	:= OUT_22_DOH;			(* Клапан софт-стоп FAN Drive	МИ-3	*)
	(*DOH_STOP_DIESEL			:	UDINT	:= OUT_24_DOH;			(* Глушение дизеля 						*)*)
	DOH_WORK_MODE_3			:	UDINT :=	OUT_25_DOH;			(* Управление планированием	в режиме бульдозера МИ-3*)


	DOH_Swim_Lamp				:	UDINT	:= OUT_21_DOH;			(* Лампа "Плавающего" режима			МИ-2*)
	DOH_FAN_Lamp				:	UDINT	:=	OUT_22_DOH;			(* Лампа режима FAN Drive 				МИ-2*)
	DOH_LOW_PRESS				:	UDINT	:= OUT_24_DOH;			(* Низкое давления растормаживания	МИ-2*)
	DOH_ERR_LAMP				:	UDINT	:= OUT_25_DOH;			(* Лампа "Ошибка" трансмиссии 		МИ-2*)
(*END_IF*)
(******************** 	Analog Outputs 				*************************************)
	AOV_KAD_RPM					:	UDINT := OUT_47_AOV;			(* Сигнал о требуемых оборотах для КАД *)


END_STRUCT
END_TYPE

(* Data type in 20_CAN/20_J1939 *)
TYPE struc_J1939 :
	STRUCT
		Box						:	struc_J1939_Box;   							(*structure to define the databox-numbers*)
		PGN						:	struc_J1939_PGN;								(*structure to define the PGN *)
		SOURCE_ADRESS			: 	USINT 							:= 0;			(*source addr - diesel usually has address "0" *)
		TIMEOUT					: 	struc_J1939_Timeout;							(*structure to define timeout of the J1939 message  *)
		Length					:	struc_J1939_DataLength; 					(*structure to define length of the J1939 message  *)
		Data						:	struc_J1939_Data;								(*data structure of the J1939 message content *)
		DISABLE_CALLBACK		: 	UINT 								:= 16#FFFF;	(*No callback functions defined, "j1939_getRxDataboxStatus" shoul be used instead*)
		Status					: 	struc_CAN_Status;   							(* structure to define the J1939 databox status *)
	END_STRUCT
END_TYPE

(* Data type in 20_CAN/20_J1939 *)
TYPE struc_J1939_Box :
	STRUCT
		Tx_TSC1_u16			:	UINT	:= 2;
		Tx_VF					:	UINT	:= 3;		(* *)
		Tx_TRF2				:	UINT	:= 4;		(* *)
		Tx_MP					:	UINT	:= 5;		(*	*)
		Tx_ESSI				:	UINT	:= 6;		(* *)
		Tx_HOURS				:	UINT	:= 7;
		Tx_EEC1				:	UINT	:= 8;
		Tx_BJM1				:	UINT	:= 9;		(* *)
 		Tx_TF_u16			:	UINT	:= 10;
 		Tx_ETC2_u16			:	UINT	:= 11;
		Tx_TFAC_u16			:	UINT	:= 12;
		Tx_RHS				:	UINT	:= 13;		(* *)
		Tx_LOI				:	UINT	:= 14;		(* *)
		Tx_ET1				:	UINT	:= 15;
		Tx_AV00MF			:	UINT	:= 16;		(* *)
		Tx_AV01MF			:	UINT	:= 17;		(* *)
		Tx_AV02MF			:	UINT	:= 18;		(* *)
		Tx_AV03MF			:	UINT	:= 19;		(* *)
		Tx_AV04MF			:	UINT	:= 20;		(* *)
(******************************************************************************)
(******************** Definition: databoxes Rx J1939*************************)
(******************************************************************************)
		Rx_EEC1_u16			:	UINT	:= 2;	(*databox to receive values from the customer*)
 		(*Rx_EEC2_u16			:	UINT	:= 3;	(*databox to receive values from the customer*)
 		Rx_EEC3_u16			:	UINT	:= 4;	(*databox to receive values from the customer*)*)
 		Rx_ET1_u16			:	UINT	:= 3;	(*databox to receive values from the customer*)
 		Rx_IC1_u16			:	UINT	:= 4;	(*databox to receive values from the customer*)
		Rx_EFL_u16			:	UINT	:= 5;
		Rx_DD_u16			:	UINT	:= 6;	(* Dash Display *)
		Rx_DIESEL_DM1_u16	:	UINT	:=	7;	(* сообщение DM1 контроллера двигателя *)
		Rx_DIESEL_DM2_u16	:	UINT	:=	8;	(* сообщение DM2 контроллера двигателя *)
	END_STRUCT
END_TYPE
		(*Tx_DM1_u16			:	UINT	:= 12;*)
 		(*Tx_StTransm_u16		:	UINT	:= 15;*)

(* Data type in 20_CAN/20_J1939 *)
TYPE struc_J1939_Data :
	STRUCT
	(* @CAN *)
  (*CAN1_Rx_buf				: ARRAY [1..43] OF can_Message_ts;		(* can receive buffer - NOT NEEDED AS in BD is DONE BY API!	*)
  CAN1_Tx_buf				: ARRAY [1..43] OF can_Message_ts;		(* can send buffer  	- NOT NEEDED AS in BD is DONE BY API! *)*)

		j1939_RxMsg_as			:	ARRAY [1..8]	OF j1939_rxMsg_ts;		(* j1939 rx msg boxes *)
		j1939_TxMsg_as			:	ARRAY [1..20]	OF j1939_txMsg_ts;		(* j1939 tx msg boxes *)

		RxEEC1_au8 				:	ARRAY [1..8] OF USINT;   (* data buffer for j1939 rx message 1 *)
 		(*RxEEC2_au8 				:	ARRAY [1..8] OF USINT;   (* data buffer for j1939 rx message 2 *)
 		RxEEC3_au8 				:	ARRAY [1..8] OF USINT;   (* data buffer for j1939 rx message 3 *)*)
		RxET1_au8  				:	ARRAY [1..8] OF USINT;   (* data buffer for j1939 rx message 1 *)
		RxIC1_au8  				:	ARRAY [1..8] OF USINT;   (* data buffer for j1939 rx message 1 *)
		RxEFL_au8 				:	ARRAY [1..8] OF USINT;
		RxDD_au8					:	ARRAY [1..8] OF USINT;

		TxBJM1					:	ARRAY [1..8] OF USINT;	(**)
		TxVF						:	ARRAY [1..8] OF USINT;	(**)
		TxTRF2					:	ARRAY [1..8] OF USINT;	(**)
		TxMP						:	ARRAY [1..8] OF USINT;	(**)
		TxESSI					:	ARRAY [1..8] OF USINT;	(**)
		TxHOURS					:	ARRAY [1..8] OF USINT;	(**)
		TxEEC1					:	ARRAY [1..8] OF USINT;
		TxRHS						:	ARRAY [1..8] OF USINT;	(**)
		TxLOI						:	ARRAY [1..8] OF USINT;	(**)
		TxET1						:	ARRAY [1..8] OF USINT;	(**)
		TxTSC1_au8 				:	ARRAY [1..8] OF USINT;
 		TxETC2_au8 				:	ARRAY [1..8] OF USINT;
 		TxTF_au8   				:	ARRAY [1..8] OF USINT;
		TxTFAC_au8				:	ARRAY [1..8] OF USINT;	(* data for actuator Thomson *)
		TxAV00MF					:	ARRAY [1..8] OF USINT;	(**)
		TxAV01MF					:	ARRAY [1..8] OF USINT;	(**)
		TxAV02MF					:	ARRAY [1..8] OF USINT;	(**)
		TxAV03MF					:	ARRAY [1..8] OF USINT;	(**)
		TxAV04MF					:	ARRAY [1..8] OF USINT;	(**)
	END_STRUCT
END_TYPE
 		(*TxStTransm_au8			:	ARRAY [1..8] OF USINT;*)

(* Data type in 20_CAN/20_J1939 *)
TYPE struc_J1939_DataLength :
	STRUCT
		J1939_STD_MSG_LEN	: 	UINT	:= 8;
		(* Нужно проверить можно ли использовать одну переменную вместо следующих *)
		EEC1					: 	UINT	:= 8;
		(*EEC2					:	UINT	:= 8;
 		EEC3					: 	UINT	:= 8;*)
		EFL_u16				:	UINT	:= 8;
		ET1_u16				:	UINT	:= 8;
		IC1_u16				:	UINT	:= 8;

		OFFSET_0				:	UINT	:= 0;
		OFFSET_10			:	UINT	:= 10;
		OFFSET_20			:	UINT	:= 20;

		PRIOR_DEFAULT		:	USINT	:= 6;
		PRIOR_3				:	USINT	:= 3;

		CYCLE_TSC1			:	UINT	:= 10;
		CYCLE_TFAC			:	UINT	:= 50;
		CYCLE_DEFAULT		:	UINT	:= 100;
		CYCLE_LOCARUS		:	UINT	:= 200;
		CYCLE_DM1			:	UINT	:= 1000;

		SA_Req_PGN			:	DWORD;					(* Source Address для запроса PGN *)
		SA_DM2_DM3_YAMZ	:	DWORD := 16#21;		(* Source Address для запроса PGN у двигателя ЯМЗ *)
		SA_DM2_CUMMINS		:	DWORD := 16#FF;		(* Source Address для запроса сохраненных ошибок у двигателя Cummins *)
		SA_DM3_CUMMINS		:	DWORD := 16#27;		(* Source Address для запроса на удаление сохраненных ошибок у двигателя Cummins *)

		Rx_DM1_Diesel_u16	:	UINT	;
		Rx_DM2_Diesel_u16	:	UINT	;

	(*	TFAC				: 	UINT	:= 8;
		BJM1				:	UINT	:= 8;
		AV00MF			:	UINT	:= 8;
		AV01MF			:	UINT	:= 8;
		VF					:	UINT	:= 8;
		TRF2				:	UINT	:= 8;
		CCVS				:	UINT	:= 8;
		MP					:	UINT	:= 8;
		ESSI				:	UINT	:= 8;*)
	END_STRUCT
END_TYPE

(* Data type in 20_CAN/20_J1939 *)
TYPE struc_J1939_PGN :
STRUCT

(******************************************************************************)
(******************** Definition: CAN IDs  ************************************)
(******************************************************************************)
	EEC1:					DWORD 	:= 16#F004;
	(*EEC2:					DWORD 	:= 16#F003;	(* Пересмотреть: нужна ли эта посылка? *)
	EEC3:					DWORD 	:= 16#FEDF;	(* Пересмотреть: нужна ли эта посылка? *)*)
	TSC1:					DWORD 	:= 16#0000;
	ET1_u32:				DWORD 	:= 16#FEEE;
	IC1_u32:				DWORD 	:= 16#FEF6;
	TF_u32:				DWORD 	:= 16#FEF8; (* Transmission Fluids - Oil Temperature in Tank *)
	ETC2_u32:			DWORD 	:= 16#F005; (* Electronic Transmission Controller - FNR/Gear Status,Brakes..*)
	TFAC:					DWORD		:= 16#F01A;	(*  *)
	EFL_u32:				DWORD		:= 16#FEEF;
	BJM1:					DWORD		:= 16#FDD6;
	VF:					DWORD		:= 16#FE68;
	TRF2:					DWORD		:= 16#FD95;
	MP:					DWORD		:= 16#FE47;
	ESSI:					DWORD		:= 16#F021;
	HOURS:				DWORD		:= 16#FEE5;
	RHS:					DWORD		:= 16#FE45;	(* Индикация работы задним навесным оборудованием - Rear Hitch In-work Indication, SPN - 1877 *)
	LOI:					DWORD		:= 16#F00D;	(* Индикация "плавающего" режима - Blade Control Mode Switch, SPN - 3156 *)
	AV00MF:				DWORD		:= 16#FE20;
	AV01MF:				DWORD		:= 16#FE21;
	AV02MF:				DWORD		:= 16#FE22;	(* Давление в контуре навесного оборудования + давление в контуре Фан-драйв *)
	AV03MF:				DWORD		:= 16#FE23;	(* Ошибки 1 *)
	AV04MF:				DWORD		:= 16#FE24;	(* Ошибки 2, 3 *)
	DD:					DWORD		:= 16#FEFC;	(* Dash Display, уровень топлива *)

	(*Modem_201:			DWORD		:= 16#0201;
	Modem_202:			DWORD		:= 16#0202;
	Modem_203:			DWORD		:= 16#0203;
	Modem_204:			DWORD		:= 16#0204;
	Modem_205:			DWORD		:= 16#0205;
	Modem_206:			DWORD		:= 16#0206;
	Modem_207:			DWORD		:= 16#0207;
	Modem_208:			DWORD		:= 16#0208;
	Modem_209:			DWORD		:= 16#0209;
	Modem_210:			DWORD		:= 16#0210;
	Modem_211:			DWORD		:= 16#0211;
	Modem_212:			DWORD		:= 16#0212;
	Modem_213:			DWORD		:= 16#0213;
	Modem_214:			DWORD		:= 16#0214;
	Modem_215:			DWORD		:= 16#0215;
	Modem_216:			DWORD		:= 16#0216;

	MI3_220:				DWORD		:= 16#0220;
	MI3_221:				DWORD		:= 16#0221;

	Modem_300:			DWORD		:= 16#0300;

	Modem_401:			DWORD		:= 16#0401;
	Modem_402:			DWORD		:= 16#0402;*)
	(*StTransm_u32:		DWORD		:= 16#FF00; (* Transm Emergency - Low Pressure / Filter Contamination*)*)
	(*CCVS:					DWORD		:= 16#FEF1;*)
	(*FD:					DWORD		:= 16#FEBD;	(* Fan Drive *)*)
END_STRUCT
END_TYPE

(* Data type in 20_CAN/20_J1939 *)
TYPE struc_J1939_Timeout :
	STRUCT
		EEC1				:	UINT	:= 1000;		(*J1939 timeout, ms*)
		(*EEC2				:	UINT	:= 1000;
		EEC3				:	UINT	:= 1000;*)
		ET1_u16			:	UINT	:= 1000;
		IC1_u16			:	UINT	:= 1000;
		TFAC				:	UINT	:= 50;
		TSC1				:	UINT	:= 50;
		EFL_u16			:	UINT	:= 1000;
		DD_timeout		:	UINT	:= 1000;
	END_STRUCT
END_TYPE

(* Data type in 10_IO *)
TYPE struc_outputs :
STRUCT  (* VL 14/03-2012 - complete this part according to req. *)

	iAct_Out_01_ma_s32			: DINT;		(* Actual current, Unit = mA *)
	iAct_Out_02_ma_s32			: DINT;		(* Actual current, Unit = mA *)
	iAct_Out_03_ma_s32			: DINT;		(* Actual current, Unit = mA *)
	iAct_Out_04_ma_s32			: DINT;		(* Actual current, Unit = mA *)
	iAct_Out_05_ma_s32			: DINT;		(* Actual current, Unit = mA *)
	iAct_Out_06_ma_s32			: DINT;		(* Actual current, Unit = mA *)
	iAct_Out_07_ma_s32			: DINT;		(* Actual current, Unit = mA *)
	iAct_Out_08_ma_s32			: DINT;		(* Actual current, Unit = mA *)
	iAct_Out_09_ma_s32			: DINT;		(* Actual current, Unit = mA *)
	iAct_Out_10_ma_s32			: DINT;		(* Actual current, Unit = mA *)
	iAct_Out_11_ma_s32			: DINT;		(* Actual current, Unit = mA *)
	iAct_Out_12_ma_s32			: DINT;		(* Actual current, Unit = mA *)
	iAct_Out_13_ma_s32			: DINT;		(* Actual current, Unit = mA *)
	iAct_Out_14_ma_s32			: DINT;		(* Actual current, Unit = mA *)
	iAct_Out_15_ma_s32			: DINT;		(* Actual current, Unit = mA *)
	iAct_Out_16_ma_s32			: DINT;		(* Actual current, Unit = mA *)
	iAct_Out_17_ma_s32			: DINT;		(* Actual current, Unit = mA *)
	iAct_Out_18_ma_s32			: DINT;		(* Actual current, Unit = mA *)
	iAct_Out_19_ma_s32			: DINT;		(* Actual current, Unit = mA *)
	iAct_Out_20_ma_s32			: DINT;		(* Actual current, Unit = mA *)
	iAct_Out_21_ma_s32			: DINT;		(* Actual current, Unit = mA *)
	iAct_Out_22_ma_s32			: DINT;		(* Actual current, Unit = mA *)
	iAct_Out_23_ma_s32			: DINT;		(* Actual current, Unit = mA *)
	iAct_Out_24_ma_s32			: DINT;		(* Actual current, Unit = mA *)
	iAct_Out_25_ma_s32			: DINT;		(* Actual current, Unit = mA *)
	iAct_Out_26_ma_s32			: DINT;		(* Actual current, Unit = mA *)
	iAct_Out_27_ma_s32			: DINT;		(* Actual current, Unit = mA *)
	iAct_Out_28_ma_s32			: DINT;		(* Actual current, Unit = mA *)
	iAct_Out_29_ma_s32			: DINT;		(* Actual current, Unit = mA *)
	iAct_Out_30_ma_s32			: DINT;		(* Actual current, Unit = mA *)
	iAct_Out_31_ma_s32			: DINT;		(* Actual current, Unit = mA *)
	iAct_Out_32_ma_s32			: DINT;		(* Actual current, Unit = mA *)
	iAct_Out_37_ma_s32			: DINT;		(* Actual current, Unit = mA *)
	iAct_Out_38_ma_s32			: DINT;		(* Actual current, Unit = mA *)
	iAct_Out_39_ma_s32			: DINT;		(* Actual current, Unit = mA *)
	iAct_Out_40_ma_s32			: DINT;		(* Actual current, Unit = mA *)
	iAct_Out_41_ma_s32			: DINT;		(* Actual current, Unit = mA *)
	iAct_Out_42_ma_s32			: DINT;		(* Actual current, Unit = mA *)
	iAct_Out_43_ma_s32			: DINT;		(* Actual current, Unit = mA *)
	iAct_Out_44_ma_s32			: DINT;		(* Actual current, Unit = mA *)
	iAct_Out_45_ma_s32			: DINT;		(* Actual current, Unit = mA *)
	iAct_Out_46_ma_s32			: DINT;		(* Actual current, Unit = mA *)


	out_01_s							: out_ts;	(* Structure with extended output information *)
	out_02_s							: out_ts;	(* Structure with extended output information *)
	out_03_s							: out_ts;	(* Structure with extended output information *)
	out_04_s							: out_ts;	(* Structure with extended output information *)
	out_05_s							: out_ts;	(* Structure with extended output information *)
	out_06_s							: out_ts;	(* Structure with extended output information *)
	out_07_s							: out_ts;	(* Structure with extended output information *)
	out_08_s							: out_ts;	(* Structure with extended output information *)
	out_09_s							: out_ts;	(* Structure with extended output information *)
	out_10_s							: out_ts;	(* Structure with extended output information *)
	out_11_s							: out_ts;	(* Structure with extended output information *)
	out_12_s							: out_ts;	(* Structure with extended output information *)
	out_13_s							: out_ts;	(* Structure with extended output information *)
	out_14_s							: out_ts;	(* Structure with extended output information *)
	out_15_s							: out_ts;	(* Structure with extended output information *)
	out_16_s							: out_ts;	(* Structure with extended output information *)
	out_17_s							: out_ts;	(* Structure with extended output information *)
	out_18_s							: out_ts;	(* Structure with extended output information *)
	out_19_s							: out_ts;	(* Structure with extended output information *)
	out_20_s							: out_ts;	(* Structure with extended output information *)
	out_21_s							: out_ts;	(* Structure with extended output information *)
	out_22_s							: out_ts;	(* Structure with extended output information *)
	out_23_s							: out_ts;	(* Structure with extended output information *)
	out_24_s							: out_ts;	(* Structure with extended output information *)
	out_25_s							: out_ts;	(* Structure with extended output information *)
	out_26_s							: out_ts;	(* Structure with extended output information *)
	out_27_s							: out_ts;	(* Structure with extended output information *)
	out_28_s							: out_ts;	(* Structure with extended output information *)
	out_29_s							: out_ts;	(* Structure with extended output information *)
	out_30_s							: out_ts;	(* Structure with extended output information *)
	out_31_s							: out_ts;	(* Structure with extended output information *)
	out_32_s							: out_ts;	(* Structure with extended output information *)
	out_33_s							: out_ts;	(* Structure with extended output information *)
	out_34_s							: out_ts;	(* Structure with extended output information *)
	out_35_s							: out_ts;	(* Structure with extended output information *)
	out_36_s							: out_ts;	(* Structure with extended output information *)
	out_37_s							: out_ts;	(* Structure with extended output information *)
	out_38_s							: out_ts;	(* Structure with extended output information *)
	out_39_s							: out_ts;	(* Structure with extended output information *)
	out_40_s							: out_ts;	(* Structure with extended output information *)
	out_41_s							: out_ts;	(* Structure with extended output information *)
	out_42_s							: out_ts;	(* Structure with extended output information *)
	out_43_s							: out_ts;	(* Structure with extended output information *)
	out_44_s							: out_ts;	(* Structure with extended output information *)
	out_45_s							: out_ts;	(* Structure with extended output information *)
	out_46_s							: out_ts;	(* Structure with extended output information *)
	out_47_s							: out_ts;	(* Structure with extended output information *)


END_STRUCT
END_TYPE

(* Data type in UDS *)
TYPE struc_Uds :
	STRUCT
		UdsRx      : struc_Uds_rx;
		UdsTx      : struc_Uds_tx;
		status     : USINT;
		initDone   : USINT;
		sessionType : USINT;
		activeAccessLevel_u8 : USINT;
		tester : UINT;
	END_STRUCT
END_TYPE

(* Data type in UDS *)
TYPE struc_Uds_rx :
	STRUCT
		dataSize : USINT;
		data     : ARRAY[1..256] OF USINT;
	END_STRUCT
END_TYPE

(* Data type in UDS *)
TYPE struc_Uds_tx :
	STRUCT
		dataSize : USINT;
		data     : ARRAY[1..256] OF USINT;
	END_STRUCT
END_TYPE

(* POU PLC_PRG, ST *)
PROGRAM PLC_PRG
VAR
(* program name and version number *)
	stSysInit_u16: 		UINT;											(* State of Sys_init(...) *)
(* В названии ПО обязательно оставить формат '*v0.00.0' -> при изменении названия ПО ознакомиться с ограничениями в get_Software_name() *)
	SW_Name_as8: 			STRING(32) := 'Laboratory_Stand';	(* Software Name *)
(*	HW_Name_as8: 			STRING(32) := 'RC30-02D6';  *)		(* RC12-10/30 Hardware Name *)
	HW_Name_as8: 			STRING(32) := 'RC30-00D6';  			(* RC28-14/30 Hardware Name *)

(* task definition *)
	MAIN_Task_Handle_u8:	USINT;		(* Task Handler for future reference e.g. checkpoint,duration, .. *)
	stMAIN_Task_u16: 		UINT;			(* State of Sys_registerTask(...) *)
	stEMCY_u16: 			UINT;
	EcuInfo_s: 				EcuInfo_ts;	(* Информация о контроллере *)
	stUds: UINT;

	POH_CL_RESISTANCE_MIN			: UDINT	:= 2000; 			(* min resistance of solenoid for error detection [mOhm]*)
	POH_CL_RESISTANCE_MAX			: UDINT	:= 52000;			(* max resistance of solenoid for error detection[mOhm] *)
	POL_CL_RESISTANCE_MIN			: UDINT	:= 2000; 			(* min resistance of solenoid for error detection [mOhm]*)
	POL_CL_RESISTANCE_MAX			: UDINT	:= 52000;			(* max resistance of solenoid for error detection[mOhm] *)
	DOH_RESISTANCE_MIN				: UDINT	:= 6000;				(* min resistance of solenoid for error detection [mOhm]*)
	DOH_RESISTANCE_MAX				: UDINT	:= 44000;			(* max resistance of solenoid for error detection[mOhm] *)
	AOV_RESISTANCE_MIN				: UDINT	:= 0; 				(* min resistance of solenoid for error detection [mOhm]*)
	AOV_RESISTANCE_MAX				: UDINT	:= 0;					(* max resistance of solenoid for error detection[mOhm] *)
	AOC_RESISTANCE_MIN				: UDINT	:= 0; 				(* min resistance of solenoid for error detection [mOhm]*)
	AOC_RESISTANCE_MAX				: UDINT	:= 0;					(* max resistance of solenoid for error detection[mOhm] *)
END_VAR

VAR CONSTANT
(******************************************************************************)
(******************** Definition:   analog input 10 V  ************************)
(******************************************************************************)
	AIV_10V_LEVEL_LOW:	INT := 4000;	(* low *)
	AIV_10V_LEVEL_HIGH:	INT := 6000;	(* high *)
	AIV_10V_DELAY:			INT := 100;		(* delay *)
	AIV_10V_ERROR_LOW:	INT := 1000;	(* low_error *)
	AIV_10V_ERROR_HIGH:	INT := 9000;	(* high_error *)
	AIV_10V_ERROR_DELAY:	INT := 100;		(* delay_error *)
(******************************************************************************)
(******************** Definition:   analog input 5V  **************************)
(******************************************************************************)
	AIV_5V_LEVEL_LOW:		INT := 2000;	(* low *)
	AIV_5V_LEVEL_HIGH:	INT := 3000;	(* high *)
	AIV_5V_DELAY:			INT := 100;		(* delay *)
	AIV_5V_ERROR_LOW:		INT := 400;		(* low_error *)
	AIV_5V_ERROR_HIGH:	INT := 4600;	(* high_error *)
	AIV_5V_ERROR_DELAY:	INT := 100;		(* delay_error *)
(******************************************************************************)
(******************** Definition:   input group  ******************************)
(******************************************************************************)
	GRP_IN1_IN8: 				USINT := 1;
	GRP_IN9_IN14: 				USINT := 2;
	GRP_IN15_IN20: 			USINT := 3;
(******************************************************************************)
	HW_Type_RC12_10_30_u16: UINT	:= 16#02D6;
END_VAR
(******************** definition: SW name and HW name *************************)
stSysInit_u16 := sys_init( ADR( SW_Name_as8 ), ADR( HW_Name_as8 ) );

(******************** definition: task   **************************************)
(* main task *)
stMAIN_Task_u16 := sys_registerTask( INDEXOF(Callback_MAIN_Task),
											 MAIN_TASK_PRIO,
											 CYCLE,
											 0,
											 ADR( MAIN_Task_Handle_u8 ));

stUds := sys_registerTask( INDEXOF(UDS_Task),
									4,
									5,
									0,
									0);
(* Set trigger checkpoint for above task *)
sys_initTC(	MAIN_Task_Handle_u8, 	CYCLE );

(* register callback function for parameters *)
diag_setVarsCallBack( INDEXOF( Callback_update_appl_param ) );
(* load all parameters when starting up *)
Callback_update_appl_param();

(*PrmData_Sample();*)
PrmData();
ProcData();
UnitCodes();
Lists();
ErrorsList();
(* Load SW information *)
SW_Version();
SwInfo();
(******************** Configuration:Sensor supply  ****************************)
(*By RC28-14 is VSS1 always ON*)
sys_setVSS( VSS_2, ON );		(* 10 V @ RC12-10 *)
sys_setVSS( VSS_3, ON );		(* 5V @ RC12-10 *)

(* Получение информации о контроллере *)
sys_getEcuInfo(ADR(EcuInfo_s));

PLC_initCAN();
PLC_initJ1939();
PLC_cfgInputs();
PLC_cfgOutputs();

(* disable the software INHIBIT *)
(* This command is necessary if pin 112 shall be used as input and not as software INH input *)
stEMCY_u16 := emcy_disableInput(EMCY_DISABLE_KEY_DU32, NOT UDINT_TO_DWORD(EMCY_DISABLE_KEY_DU32));
END_PROGRAM
ACTION PLC_cfgInputs:
(*TO BE REMOVED******************************************************************************
It is recommended to initialize all input channels
This ensures that a possible change of the RTS will not affect the settings 

The initialization of an input signal requires the following steps :
- Configuration of the internal pullup/pulldown (in_setPullup)
- Definition of the channel name (see  Global_Channels (CONSTANT) )
- A monitoring process (in_cfgVoltageInput)
- for a potentiometer: a definition of a voltage range (inext_cfgPoti)  
********************************************************************************************)

(*******************************************************************************************)
(******************** @IN_PUMP: configuration of the desired swivel angle for the pump *****)
(*******************************************************************************************)

(**********************)
(* With INEXT Library *)
(**********************)
 inext_cfgPoti(IO_Chnl.AI_JOY_DRIVE, MAX_VOLTAGE_FOR_JOY);			(* Define a 5 V maximum voltage in mV *)
 inext_cfgPoti(IO_Chnl.AI_JOY_STEER, MAX_VOLTAGE_FOR_JOY);			(* Define a 5 V maximum voltage in mV *)
 inext_cfgPoti(IO_Chnl.AI_POTI_DIESEL, 5000);							(* Define a 5 V maximum voltage in mV *)
 inext_cfgPoti(IO_Chnl.AI_BRAKE_PEDAL, 5000);							(* Define a 5 V maximum voltage in mV *)

 inext_cfgPoti(IO_Chnl.AI_BOM_SPEED, 5000);								(* Define a 5 V maximum voltage in mV *)

 inext_cfgPoti(IO_Chnl.AI_JOY_DIRECTION, MAX_VOLTAGE_FOR_JOY);
 inext_cfgPoti(IO_Chnl.AI_JOY_SIDE, MAX_VOLTAGE_FOR_JOY);

(* Configure the inputs 54 - 61 for current mesurement *)
in_setCurrentMeasurement(2, ON);
(*in_setCurrentMeasurement(3, ON);*)

in_cfgCurrentInput( IO_Chnl.AI_JOY_DRIVE_CM, DOH_DEBOUNCE);
in_cfgCurrentInput( IO_Chnl.AI_JOY_STEER_CM, DOH_DEBOUNCE);
(*in_cfgCurrentInput( IO_Chnl.AI_JOY_DIRECTION_CM, DOH_DEBOUNCE);
in_cfgCurrentInput( IO_Chnl.AI_JOY_SIDE_CM, DOH_DEBOUNCE);*)

(*
in_cfgCurrentInput( IO_Chnl.AI_POTI_DIESEL_CM, DOH_DEBOUNCE);	(* Добавлено 23.10.15 Для работы бесконтактного датчика *)
in_cfgCurrentInput( IO_Chnl.AI_BRAKE_PEDAL_CM, DOH_DEBOUNCE);	(* Добавлено 23.10.15 Для работы бесконтактного датчика *)
*)
(************************************************************)
(*
in_cfgTempSensorType(IO_Chnl.AIT_OIL_TEMP_TANK, 1);
*)
(*
in_cfgVoltageInput( 	IO_Chnl.AI_BRAKE_PEDAL,				(*chnl*)
							AIV_5V_LEVEL_LOW,				(*low*)
							AIV_5V_LEVEL_HIGH,			(*high*)
							AIV_5V_DELAY,					(*delay*)
							AIV_5V_ERROR_LOW,				(*low_error*)
							AIV_5V_ERROR_HIGH,			(*high_error*)
							AIV_5V_ERROR_DELAY );		(*delay_error*)


(*******************************************************************************************)
(******************** @IN_INCH: configuration of the inch pedal signal (max voltage: 5V)****)
(*******************************************************************************************)
in_cfgVoltageInput( 	IO_Chnl.AI_MOTOR_R_SIMUL,				(*chnl*)
							AIV_10V_LEVEL_LOW,			(*low*)
							AIV_10V_LEVEL_HIGH,			(*high*)
							AIV_10V_DELAY,					(*delay*)
							AIV_10V_ERROR_LOW,			(*low_error*)
							AIV_10V_ERROR_HIGH,			(*high_error*)
							AIV_10V_ERROR_DELAY );		(*delay_error*)
*)

(*
2nd alternative representation:
-------------------------------
*)  
(*
(* in_cfgVoltageInput ( chnl_u32, uLowerStateThreshold_s16, uUpperStateThreshold_s16,
tiStateDebounce_s16, uLowerDiagThreshold_s16, uUpperDiagThreshold_s16, tiDiagDebounce_s16 ) *)
in_cfgVoltageInput( 	IO_Chnl.AIV_INCH,	4000,	6000,	100,	1000,	9000,	100);
in_cfgVoltageInput( 	IO_Chnl.AIV_PUMP,	2000,	3000,	100,	400,	4600,	100);
*)

(*******************************************************************************************)
(******************** @IN_DIESEL: configuration of the actual speed of the diesel **********)
(*******************************************************************************************)
(*no initialisation expected*)

(*******************************************************************************************)
(************* @IN_DRIVE_SPEED_ACTUAL:  configuration of the actual speed of the vehicle **)
(*******************************************************************************************)
(*no initialisation expected*)

(*******************************************************************************************)
(******************** @IN_BRAKE: configuration of the parking brake switch *****************)
(*******************************************************************************************)
(*no initialisation expected*)
END_ACTION
ACTION PLC_cfgOutputs:
POH_CL_RESISTANCE_MIN			:= (para_s.POH_Res_Min_s16*1000);
POH_CL_RESISTANCE_MAX			:= (para_s.POH_Res_Max_s16*1000);
DOH_RESISTANCE_MIN				:= (para_s.DOH_Res_Min_s16*1000);
DOH_RESISTANCE_MAX				:= (para_s.DOH_Res_Max_s16*1000);
POL_CL_RESISTANCE_MIN			:= (para_s.POL_Res_Min_s16*1000);
POL_CL_RESISTANCE_MAX			:= (para_s.POL_Res_Max_s16*1000);
AOV_RESISTANCE_MIN				:= (para_s.AOV_Res_Min_s16*1000);
AOV_RESISTANCE_MAX				:= (para_s.AOV_Res_Max_s16*1000);
AOC_RESISTANCE_MIN				:= (para_s.AOC_Res_Min_s16*1000);
AOC_RESISTANCE_MAX				:= (para_s.AOC_Res_Max_s16*1000);
(******************************************************************************************************)
(* Proportional Output High *)
(******************************************************************************************************)

IF para_s.Out_Cfg_01_s16 = PWM_MODE THEN
	out_cfg	(	OUT_1_POH,							(* PWM output close loop *)
					para_s.POH_Debounce_s16,		(* debounce time [ms] for error detection *)
					POH_CL_DITHER_FREQUENCY, 		(* dither frequency [Hz] *)
					POH_CL_RESISTANCE_MIN, 			(* min resistance of solenoid for error detection [mOhm]*)
					POH_CL_RESISTANCE_MAX );		(* max resistance of solenoid for error detection[mOhm] *)
ELSIF para_s.Out_Cfg_01_s16 = PWM_CURRENT_MODE THEN
	out_cfg	(	OUT_1_POH_CL,						(* PWM output close loop *)
					para_s.POH_Debounce_s16,		(* debounce time [ms] for error detection *)
					POH_CL_DITHER_FREQUENCY, 		(* dither frequency [Hz] *)
					POH_CL_RESISTANCE_MIN, 			(* min resistance of solenoid for error detection [mOhm]*)
					POH_CL_RESISTANCE_MAX );		(* max resistance of solenoid for error detection[mOhm] *)

	out_cfgPI(	OUT_1_POH_CL,						(*Channel*)
			      para_s.POH_Kp_s16,				(*Kp factor*)
	      		para_s.POH_Ki_s16 );				(*Ki factor*)
END_IF

IF para_s.Out_Cfg_02_s16 = PWM_MODE THEN
	out_cfg	(	OUT_2_POH,							(* PWM output close loop *)
					para_s.POH_Debounce_s16,		(* debounce time [ms] for error detection *)
					POH_CL_DITHER_FREQUENCY, 		(* dither frequency [Hz] *)
					POH_CL_RESISTANCE_MIN, 			(* min resistance of solenoid for error detection [mOhm]*)
					POH_CL_RESISTANCE_MAX );		(* max resistance of solenoid for error detection[mOhm] *)
ELSIF para_s.Out_Cfg_02_s16 = PWM_CURRENT_MODE THEN
	out_cfg	(	OUT_2_POH_CL,						(* PWM output close loop *)
					para_s.POH_Debounce_s16,		(* debounce time [ms] for error detection *)
					POH_CL_DITHER_FREQUENCY, 		(* dither frequency [Hz] *)
					POH_CL_RESISTANCE_MIN, 			(* min resistance of solenoid for error detection [mOhm]*)
					POH_CL_RESISTANCE_MAX );		(* max resistance of solenoid for error detection[mOhm] *)

	out_cfgPI(	OUT_2_POH_CL,						(*Channel*)
			      para_s.POH_Kp_s16,				(*Kp factor*)
	      		para_s.POH_Ki_s16 );				(*Ki factor*)
END_IF

IF para_s.Out_Cfg_03_s16 = PWM_MODE THEN
	out_cfg	(	OUT_3_POH,							(* PWM output close loop *)
					para_s.POH_Debounce_s16,		(* debounce time [ms] for error detection *)
					POH_CL_DITHER_FREQUENCY, 		(* dither frequency [Hz] *)
					POH_CL_RESISTANCE_MIN, 			(* min resistance of solenoid for error detection [mOhm]*)
					POH_CL_RESISTANCE_MAX );		(* max resistance of solenoid for error detection[mOhm] *)
ELSIF para_s.Out_Cfg_03_s16 = PWM_CURRENT_MODE THEN
	out_cfg	(	OUT_3_POH_CL,						(* PWM output close loop *)
					para_s.POH_Debounce_s16,		(* debounce time [ms] for error detection *)
					POH_CL_DITHER_FREQUENCY, 		(* dither frequency [Hz] *)
					POH_CL_RESISTANCE_MIN, 			(* min resistance of solenoid for error detection [mOhm]*)
					POH_CL_RESISTANCE_MAX );		(* max resistance of solenoid for error detection[mOhm] *)

	out_cfgPI(	OUT_3_POH_CL,						(*Channel*)
			      para_s.POH_Kp_s16,				(*Kp factor*)
	      		para_s.POH_Ki_s16 );				(*Ki factor*)
END_IF

IF para_s.Out_Cfg_04_s16 = PWM_MODE THEN
	out_cfg	(	OUT_4_POH,							(* PWM output close loop *)
					para_s.POH_Debounce_s16,		(* debounce time [ms] for error detection *)
					POH_CL_DITHER_FREQUENCY, 		(* dither frequency [Hz] *)
					POH_CL_RESISTANCE_MIN, 			(* min resistance of solenoid for error detection [mOhm]*)
					POH_CL_RESISTANCE_MAX );		(* max resistance of solenoid for error detection[mOhm] *)
ELSIF para_s.Out_Cfg_04_s16 = PWM_CURRENT_MODE THEN
	out_cfg	(	OUT_4_POH_CL,						(* PWM output close loop *)
					para_s.POH_Debounce_s16,		(* debounce time [ms] for error detection *)
					POH_CL_DITHER_FREQUENCY, 		(* dither frequency [Hz] *)
					POH_CL_RESISTANCE_MIN, 			(* min resistance of solenoid for error detection [mOhm]*)
					POH_CL_RESISTANCE_MAX );		(* max resistance of solenoid for error detection[mOhm] *)

	out_cfgPI(	OUT_4_POH_CL,						(*Channel*)
			      para_s.POH_Kp_s16,				(*Kp factor*)
	      		para_s.POH_Ki_s16 );				(*Ki factor*)
END_IF

IF para_s.Out_Cfg_05_s16 = PWM_MODE THEN
	out_cfg	(	OUT_5_POH,							(* PWM output close loop *)
					para_s.POH_Debounce_s16,		(* debounce time [ms] for error detection *)
					POH_CL_DITHER_FREQUENCY, 		(* dither frequency [Hz] *)
					POH_CL_RESISTANCE_MIN, 			(* min resistance of solenoid for error detection [mOhm]*)
					POH_CL_RESISTANCE_MAX );		(* max resistance of solenoid for error detection[mOhm] *)
ELSIF para_s.Out_Cfg_05_s16 = PWM_CURRENT_MODE THEN
	out_cfg	(	OUT_5_POH_CL,						(* PWM output close loop *)
					para_s.POH_Debounce_s16,		(* debounce time [ms] for error detection *)
					POH_CL_DITHER_FREQUENCY, 		(* dither frequency [Hz] *)
					POH_CL_RESISTANCE_MIN, 			(* min resistance of solenoid for error detection [mOhm]*)
					POH_CL_RESISTANCE_MAX );		(* max resistance of solenoid for error detection[mOhm] *)

	out_cfgPI(	OUT_5_POH_CL,						(*Channel*)
			      para_s.POH_Kp_s16,				(*Kp factor*)
	      		para_s.POH_Ki_s16 );				(*Ki factor*)
END_IF

IF para_s.Out_Cfg_06_s16 = PWM_MODE THEN
	out_cfg	(	OUT_6_POH,							(* PWM output close loop *)
					para_s.POH_Debounce_s16,		(* debounce time [ms] for error detection *)
					POH_CL_DITHER_FREQUENCY, 		(* dither frequency [Hz] *)
					POH_CL_RESISTANCE_MIN, 			(* min resistance of solenoid for error detection [mOhm]*)
					POH_CL_RESISTANCE_MAX );		(* max resistance of solenoid for error detection[mOhm] *)
ELSIF para_s.Out_Cfg_06_s16 = PWM_CURRENT_MODE THEN
	out_cfg	(	OUT_6_POH_CL,						(* PWM output close loop *)
					para_s.POH_Debounce_s16,		(* debounce time [ms] for error detection *)
					POH_CL_DITHER_FREQUENCY, 		(* dither frequency [Hz] *)
					POH_CL_RESISTANCE_MIN, 			(* min resistance of solenoid for error detection [mOhm]*)
					POH_CL_RESISTANCE_MAX );		(* max resistance of solenoid for error detection[mOhm] *)

	out_cfgPI(	OUT_6_POH_CL,						(*Channel*)
			      para_s.POH_Kp_s16,				(*Kp factor*)
	      		para_s.POH_Ki_s16 );				(*Ki factor*)
END_IF

IF para_s.Out_Cfg_07_s16 = PWM_MODE THEN
	out_cfg	(	OUT_7_POH,							(* PWM output close loop *)
					para_s.POH_Debounce_s16,		(* debounce time [ms] for error detection *)
					POH_CL_DITHER_FREQUENCY, 		(* dither frequency [Hz] *)
					POH_CL_RESISTANCE_MIN, 			(* min resistance of solenoid for error detection [mOhm]*)
					POH_CL_RESISTANCE_MAX );		(* max resistance of solenoid for error detection[mOhm] *)
ELSIF para_s.Out_Cfg_07_s16 = PWM_CURRENT_MODE THEN
	out_cfg	(	OUT_7_POH_CL,						(* PWM output close loop *)
					para_s.POH_Debounce_s16,		(* debounce time [ms] for error detection *)
					POH_CL_DITHER_FREQUENCY, 		(* dither frequency [Hz] *)
					POH_CL_RESISTANCE_MIN, 			(* min resistance of solenoid for error detection [mOhm]*)
					POH_CL_RESISTANCE_MAX );		(* max resistance of solenoid for error detection[mOhm] *)

	out_cfgPI(	OUT_7_POH_CL,						(*Channel*)
			      para_s.POH_Kp_s16,				(*Kp factor*)
	      		para_s.POH_Ki_s16 );				(*Ki factor*)
END_IF

IF para_s.Out_Cfg_08_s16 = PWM_MODE THEN
	out_cfg	(	OUT_8_POH,							(* PWM output close loop *)
					para_s.POH_Debounce_s16,		(* debounce time [ms] for error detection *)
					POH_CL_DITHER_FREQUENCY, 		(* dither frequency [Hz] *)
					POH_CL_RESISTANCE_MIN, 			(* min resistance of solenoid for error detection [mOhm]*)
					POH_CL_RESISTANCE_MAX );		(* max resistance of solenoid for error detection[mOhm] *)
ELSIF para_s.Out_Cfg_08_s16 = PWM_CURRENT_MODE THEN
	out_cfg	(	OUT_8_POH_CL,						(* PWM output close loop *)
					para_s.POH_Debounce_s16,		(* debounce time [ms] for error detection *)
					POH_CL_DITHER_FREQUENCY, 		(* dither frequency [Hz] *)
					POH_CL_RESISTANCE_MIN, 			(* min resistance of solenoid for error detection [mOhm]*)
					POH_CL_RESISTANCE_MAX );		(* max resistance of solenoid for error detection[mOhm] *)

	out_cfgPI(	OUT_8_POH_CL,						(*Channel*)
			      para_s.POH_Kp_s16,				(*Kp factor*)
	      		para_s.POH_Ki_s16 );				(*Ki factor*)
END_IF

IF para_s.Out_Cfg_09_s16 = PWM_MODE THEN
	out_cfg	(	OUT_9_POH,							(* PWM output close loop *)
					para_s.POH_Debounce_s16,		(* debounce time [ms] for error detection *)
					POH_CL_DITHER_FREQUENCY, 		(* dither frequency [Hz] *)
					POH_CL_RESISTANCE_MIN, 			(* min resistance of solenoid for error detection [mOhm]*)
					POH_CL_RESISTANCE_MAX );		(* max resistance of solenoid for error detection[mOhm] *)
ELSIF para_s.Out_Cfg_09_s16 = PWM_CURRENT_MODE THEN
	out_cfg	(	OUT_9_POH_CL,						(* PWM output close loop *)
					para_s.POH_Debounce_s16,		(* debounce time [ms] for error detection *)
					POH_CL_DITHER_FREQUENCY, 		(* dither frequency [Hz] *)
					POH_CL_RESISTANCE_MIN, 			(* min resistance of solenoid for error detection [mOhm]*)
					POH_CL_RESISTANCE_MAX );		(* max resistance of solenoid for error detection[mOhm] *)

	out_cfgPI(	OUT_9_POH_CL,						(*Channel*)
			      para_s.POH_Kp_s16,				(*Kp factor*)
	      		para_s.POH_Ki_s16 );				(*Ki factor*)
END_IF

IF para_s.Out_Cfg_10_s16 = PWM_MODE THEN
	out_cfg	(	OUT_10_POH,							(* PWM output close loop *)
					para_s.POH_Debounce_s16,		(* debounce time [ms] for error detection *)
					POH_CL_DITHER_FREQUENCY, 		(* dither frequency [Hz] *)
					POH_CL_RESISTANCE_MIN, 			(* min resistance of solenoid for error detection [mOhm]*)
					POH_CL_RESISTANCE_MAX );		(* max resistance of solenoid for error detection[mOhm] *)
ELSIF para_s.Out_Cfg_10_s16 = PWM_CURRENT_MODE THEN
	out_cfg	(	OUT_10_POH_CL,						(* PWM output close loop *)
					para_s.POH_Debounce_s16,		(* debounce time [ms] for error detection *)
					POH_CL_DITHER_FREQUENCY, 		(* dither frequency [Hz] *)
					POH_CL_RESISTANCE_MIN, 			(* min resistance of solenoid for error detection [mOhm]*)
					POH_CL_RESISTANCE_MAX );		(* max resistance of solenoid for error detection[mOhm] *)

	out_cfgPI(	OUT_10_POH_CL,						(*Channel*)
			      para_s.POH_Kp_s16,				(*Kp factor*)
	      		para_s.POH_Ki_s16 );				(*Ki factor*)
END_IF

IF para_s.Out_Cfg_11_s16 = PWM_MODE THEN
	out_cfg	(	OUT_11_POH,							(* PWM output close loop *)
					para_s.POH_Debounce_s16,		(* debounce time [ms] for error detection *)
					POH_CL_DITHER_FREQUENCY, 		(* dither frequency [Hz] *)
					POH_CL_RESISTANCE_MIN, 			(* min resistance of solenoid for error detection [mOhm]*)
					POH_CL_RESISTANCE_MAX );		(* max resistance of solenoid for error detection[mOhm] *)
ELSIF para_s.Out_Cfg_11_s16 = PWM_CURRENT_MODE THEN
	out_cfg	(	OUT_11_POH_CL,						(* PWM output close loop *)
					para_s.POH_Debounce_s16,		(* debounce time [ms] for error detection *)
					POH_CL_DITHER_FREQUENCY, 		(* dither frequency [Hz] *)
					POH_CL_RESISTANCE_MIN, 			(* min resistance of solenoid for error detection [mOhm]*)
					POH_CL_RESISTANCE_MAX );		(* max resistance of solenoid for error detection[mOhm] *)

	out_cfgPI(	OUT_11_POH_CL,						(*Channel*)
			      para_s.POH_Kp_s16,				(*Kp factor*)
	      		para_s.POH_Ki_s16 );				(*Ki factor*)
END_IF

IF para_s.Out_Cfg_12_s16 = PWM_MODE THEN
	out_cfg	(	OUT_12_POH,							(* PWM output close loop *)
					para_s.POH_Debounce_s16,		(* debounce time [ms] for error detection *)
					POH_CL_DITHER_FREQUENCY, 		(* dither frequency [Hz] *)
					POH_CL_RESISTANCE_MIN, 			(* min resistance of solenoid for error detection [mOhm]*)
					POH_CL_RESISTANCE_MAX );		(* max resistance of solenoid for error detection[mOhm] *)
ELSIF para_s.Out_Cfg_12_s16 = PWM_CURRENT_MODE THEN
	out_cfg	(	OUT_12_POH_CL,						(* PWM output close loop *)
					para_s.POH_Debounce_s16,		(* debounce time [ms] for error detection *)
					POH_CL_DITHER_FREQUENCY, 		(* dither frequency [Hz] *)
					POH_CL_RESISTANCE_MIN, 			(* min resistance of solenoid for error detection [mOhm]*)
					POH_CL_RESISTANCE_MAX );		(* max resistance of solenoid for error detection[mOhm] *)

	out_cfgPI(	OUT_12_POH_CL,						(*Channel*)
			      para_s.POH_Kp_s16,				(*Kp factor*)
	      		para_s.POH_Ki_s16 );				(*Ki factor*)
END_IF

IF para_s.Out_Cfg_13_s16 = PWM_MODE THEN
	out_cfg	(	OUT_13_POH,							(* PWM output close loop *)
					para_s.POH_Debounce_s16,		(* debounce time [ms] for error detection *)
					POH_CL_DITHER_FREQUENCY, 		(* dither frequency [Hz] *)
					POH_CL_RESISTANCE_MIN, 			(* min resistance of solenoid for error detection [mOhm]*)
					POH_CL_RESISTANCE_MAX );		(* max resistance of solenoid for error detection[mOhm] *)
ELSIF para_s.Out_Cfg_13_s16 = PWM_CURRENT_MODE THEN
	out_cfg	(	OUT_13_POH_CL,						(* PWM output close loop *)
					para_s.POH_Debounce_s16,		(* debounce time [ms] for error detection *)
					POH_CL_DITHER_FREQUENCY, 		(* dither frequency [Hz] *)
					POH_CL_RESISTANCE_MIN, 			(* min resistance of solenoid for error detection [mOhm]*)
					POH_CL_RESISTANCE_MAX );		(* max resistance of solenoid for error detection[mOhm] *)

	out_cfgPI(	OUT_13_POH_CL,						(*Channel*)
			      para_s.POH_Kp_s16,				(*Kp factor*)
	      		para_s.POH_Ki_s16 );				(*Ki factor*)
END_IF

IF para_s.Out_Cfg_14_s16 = PWM_MODE THEN
	out_cfg	(	OUT_14_POH,							(* PWM output close loop *)
					para_s.POH_Debounce_s16,		(* debounce time [ms] for error detection *)
					POH_CL_DITHER_FREQUENCY, 		(* dither frequency [Hz] *)
					POH_CL_RESISTANCE_MIN, 			(* min resistance of solenoid for error detection [mOhm]*)
					POH_CL_RESISTANCE_MAX );		(* max resistance of solenoid for error detection[mOhm] *)
ELSIF para_s.Out_Cfg_14_s16 = PWM_CURRENT_MODE THEN
	out_cfg	(	OUT_14_POH_CL,						(* PWM output close loop *)
					para_s.POH_Debounce_s16,		(* debounce time [ms] for error detection *)
					POH_CL_DITHER_FREQUENCY, 		(* dither frequency [Hz] *)
					POH_CL_RESISTANCE_MIN, 			(* min resistance of solenoid for error detection [mOhm]*)
					POH_CL_RESISTANCE_MAX );		(* max resistance of solenoid for error detection[mOhm] *)

	out_cfgPI(	OUT_14_POH_CL,						(*Channel*)
			      para_s.POH_Kp_s16,				(*Kp factor*)
	      		para_s.POH_Ki_s16 );				(*Ki factor*)
END_IF

IF para_s.Out_Cfg_15_s16 = PWM_MODE THEN
	out_cfg	(	OUT_15_POH,							(* PWM output close loop *)
					para_s.POH_Debounce_s16,		(* debounce time [ms] for error detection *)
					POH_CL_DITHER_FREQUENCY, 		(* dither frequency [Hz] *)
					POH_CL_RESISTANCE_MIN, 			(* min resistance of solenoid for error detection [mOhm]*)
					POH_CL_RESISTANCE_MAX );		(* max resistance of solenoid for error detection[mOhm] *)
ELSIF para_s.Out_Cfg_15_s16 = PWM_CURRENT_MODE THEN
	out_cfg	(	OUT_15_POH_CL,						(* PWM output close loop *)
					para_s.POH_Debounce_s16,		(* debounce time [ms] for error detection *)
					POH_CL_DITHER_FREQUENCY, 		(* dither frequency [Hz] *)
					POH_CL_RESISTANCE_MIN, 			(* min resistance of solenoid for error detection [mOhm]*)
					POH_CL_RESISTANCE_MAX );		(* max resistance of solenoid for error detection[mOhm] *)

	out_cfgPI(	OUT_15_POH_CL,						(*Channel*)
			      para_s.POH_Kp_s16,				(*Kp factor*)
	      		para_s.POH_Ki_s16 );				(*Ki factor*)
END_IF

IF para_s.Out_Cfg_16_s16 = PWM_MODE THEN
	out_cfg	(	OUT_16_POH,							(* PWM output close loop *)
					para_s.POH_Debounce_s16,		(* debounce time [ms] for error detection *)
					POH_CL_DITHER_FREQUENCY, 		(* dither frequency [Hz] *)
					POH_CL_RESISTANCE_MIN, 			(* min resistance of solenoid for error detection [mOhm]*)
					POH_CL_RESISTANCE_MAX );		(* max resistance of solenoid for error detection[mOhm] *)
ELSIF para_s.Out_Cfg_16_s16 = PWM_CURRENT_MODE THEN
	out_cfg	(	OUT_16_POH_CL,						(* PWM output close loop *)
					para_s.POH_Debounce_s16,		(* debounce time [ms] for error detection *)
					POH_CL_DITHER_FREQUENCY, 		(* dither frequency [Hz] *)
					POH_CL_RESISTANCE_MIN, 			(* min resistance of solenoid for error detection [mOhm]*)
					POH_CL_RESISTANCE_MAX );		(* max resistance of solenoid for error detection[mOhm] *)

	out_cfgPI(	OUT_16_POH_CL,						(*Channel*)
			      para_s.POH_Kp_s16,				(*Kp factor*)
	      		para_s.POH_Ki_s16 );				(*Ki factor*)
END_IF

IF para_s.Out_Cfg_17_s16 = PWM_MODE THEN
	out_cfg	(	OUT_17_POH,							(* PWM output close loop *)
					para_s.POH_Debounce_s16,		(* debounce time [ms] for error detection *)
					POH_CL_DITHER_FREQUENCY, 		(* dither frequency [Hz] *)
					POH_CL_RESISTANCE_MIN, 			(* min resistance of solenoid for error detection [mOhm]*)
					POH_CL_RESISTANCE_MAX );		(* max resistance of solenoid for error detection[mOhm] *)
ELSIF para_s.Out_Cfg_17_s16 = PWM_CURRENT_MODE THEN
	out_cfg	(	OUT_17_POH_CL,						(* PWM output close loop *)
					para_s.POH_Debounce_s16,		(* debounce time [ms] for error detection *)
					POH_CL_DITHER_FREQUENCY, 		(* dither frequency [Hz] *)
					POH_CL_RESISTANCE_MIN, 			(* min resistance of solenoid for error detection [mOhm]*)
					POH_CL_RESISTANCE_MAX );		(* max resistance of solenoid for error detection[mOhm] *)

	out_cfgPI(	OUT_17_POH_CL,						(*Channel*)
			      para_s.POH_Kp_s16,				(*Kp factor*)
	      		para_s.POH_Ki_s16 );				(*Ki factor*)
END_IF

IF para_s.Out_Cfg_18_s16 = PWM_MODE THEN
	out_cfg	(	OUT_18_POH,							(* PWM output close loop *)
					para_s.POH_Debounce_s16,		(* debounce time [ms] for error detection *)
					POH_CL_DITHER_FREQUENCY, 		(* dither frequency [Hz] *)
					POH_CL_RESISTANCE_MIN, 			(* min resistance of solenoid for error detection [mOhm]*)
					POH_CL_RESISTANCE_MAX );		(* max resistance of solenoid for error detection[mOhm] *)
ELSIF para_s.Out_Cfg_18_s16 = PWM_CURRENT_MODE THEN
	out_cfg	(	OUT_18_POH_CL,						(* PWM output close loop *)
					para_s.POH_Debounce_s16,		(* debounce time [ms] for error detection *)
					POH_CL_DITHER_FREQUENCY, 		(* dither frequency [Hz] *)
					POH_CL_RESISTANCE_MIN, 			(* min resistance of solenoid for error detection [mOhm]*)
					POH_CL_RESISTANCE_MAX );		(* max resistance of solenoid for error detection[mOhm] *)

	out_cfgPI(	OUT_18_POH_CL,						(*Channel*)
			      para_s.POH_Kp_s16,				(*Kp factor*)
	      		para_s.POH_Ki_s16 );				(*Ki factor*)
END_IF


(******************************************************************************************************)
(* Digital Output *)
(******************************************************************************************************)

	out_cfg ( 	OUT_19_DOH,
					para_s.DOH_Debounce_s16,
					f_100Hz_DU16,
					DOH_RESISTANCE_MIN,
					DOH_RESISTANCE_MAX );

	out_cfg ( 	OUT_20_DOH,
					para_s.DOH_Debounce_s16,
					f_100Hz_DU16,
					DOH_RESISTANCE_MIN,
					DOH_RESISTANCE_MAX );

	out_cfg ( 	OUT_21_DOH,
					para_s.DOH_Debounce_s16,
					f_100Hz_DU16,
					DOH_RESISTANCE_MIN,
					DOH_RESISTANCE_MAX );

	out_cfg ( 	OUT_22_DOH,
					para_s.DOH_Debounce_s16,
					f_100Hz_DU16,
					DOH_RESISTANCE_MIN,
					DOH_RESISTANCE_MAX );

